LIN {X 0,Y 249.049,Z 231.079,A -85,B 0,C 180,E1 -18869.473,E2 -18869.473} C_VEL
LIN {X 0,Y 249.067,Z 231.077,A -85,B 0,C 180,E1 -18873.162,E2 -18873.162} C_VEL
LIN {X 0,Y 249.056,Z 231.062,A -85,B 0,C 180,E1 -18876.73,E2 -18876.73} C_VEL
LIN {X 0,Y 249.103,Z 231.062,A -85,B 0,C 180,E1 -18880.211,E2 -18880.211} C_VEL
LIN {X 0,Y 249.237,Z 231.055,A -85,B 0,C 180,E1 -18883.622,E2 -18883.622} C_VEL
LIN {X 0,Y 249.239,Z 231.06,A -85,B 0,C 180,E1 -18888.616,E2 -18888.616} C_VEL
LIN {X 0,Y 249.449,Z 231.028,A -85,B 0,C 180,E1 -18891.902,E2 -18891.902} C_VEL
LIN {X 0,Y 249.291,Z 231.049,A -85,B 0,C 180,E1 -18895.149,E2 -18895.149} C_VEL
LIN {X 0,Y 249.671,Z 231.01,A -85,B 0,C 180,E1 -18898.387,E2 -18898.387} C_VEL
LIN {X 0,Y 249.671,Z 231.008,A -85,B 0,C 180,E1 -18901.613,E2 -18901.613} C_VEL
LIN {X 0,Y 249.436,Z 231.036,A -85,B 0,C 180,E1 -18906.714,E2 -18906.714} C_VEL
LIN {X 0,Y 249.339,Z 231.046,A -85,B 0,C 180,E1 -18909.737,E2 -18909.737} C_VEL
LIN {X 0,Y 249.192,Z 231.07,A -85,B 0,C 180,E1 -18914.704,E2 -18914.704} C_VEL
LIN {X 0,Y 249.13,Z 231.075,A -85,B 0,C 180,E1 -18918.078,E2 -18918.078} C_VEL
LIN {X 0,Y 249.08,Z 231.078,A -85,B 0,C 180,E1 -18921.519,E2 -18921.519} C_VEL
LIN {X 0,Y 249.113,Z 231.045,A -85,B 0,C 180,E1 -18925.476,E2 -18925.476} C_VEL
LIN {X 0,Y 249.08,Z 231.083,A -85,B 0,C 180,E1 -18928.994,E2 -18928.994} C_VEL
LIN {X 0,Y 249.027,Z 231.091,A -85,B 0,C 180,E1 -18932.427,E2 -18932.427} C_VEL
LIN {X 0,Y 249.027,Z 231.083,A -85,B 0,C 180,E1 -18936.346,E2 -18936.346} C_VEL
LIN {X 0,Y 249.031,Z 231.1,A -85,B 0,C 180,E1 -18939.615,E2 -18939.615} C_VEL
LIN {X 0,Y 249.908,Z 233.771,A -85,B 0,C 180,E1 -18939.977,E2 -18939.977} C_VEL
LIN {X 0,Y 251.817,Z 235.917,A -85,B 0,C 180,E1 -18940.589,E2 -18940.589} C_VEL
LIN {X 0,Y 252.607,Z 236.622,A -85,B 0,C 180,E1 -18940.83,E2 -18940.83} C_VEL
LIN {X 0,Y 254.612,Z 239.846,A -85,B 0,C 180,E1 -18941.489,E2 -18941.489} C_VEL
LIN {X 0,Y 256.321,Z 241.907,A -85,B 0,C 180,E1 -18942.007,E2 -18942.007} C_VEL
LIN {X 0,Y 263.064,Z 251.483,A -85,B 0,C 180,E1 -18943.997,E2 -18943.997} C_VEL
LIN {X 0,Y 271.116,Z 263.635,A -85,B 0,C 180,E1 -18946.185,E2 -18946.185} C_VEL
LIN {X 0,Y 276.17,Z 272.352,A -85,B 0,C 180,E1 -18947.494,E2 -18947.494} C_VEL
LIN {X 0,Y 283.771,Z 287.993,A -85,B 0,C 180,E1 -18949.41,E2 -18949.41} C_VEL
LIN {X 0,Y 285.944,Z 292.88,A -85,B 0,C 180,E1 -18949.943,E2 -18949.943} C_VEL
LIN {X 0,Y 281.183,Z 391.143,A -85,B 0,C 180,E1 -18952.354,E2 -18952.354} C_VEL
LIN {X 0,Y 279.713,Z 406.301,A -85,B 0,C 180,E1 -18952.971,E2 -18952.971} C_VEL
LIN {X 0,Y 277.742,Z 421.037,A -85,B 0,C 180,E1 -18953.851,E2 -18953.851} C_VEL
LIN {X 0,Y 275.453,Z 434.469,A -85,B 0,C 180,E1 -18954.923,E2 -18954.923} C_VEL
LIN {X 0,Y 272.602,Z 448.403,A -85,B 0,C 180,E1 -18956.339,E2 -18956.339} C_VEL
LIN {X 0,Y 269.202,Z 462.16,A -85,B 0,C 180,E1 -18958.086,E2 -18958.086} C_VEL
LIN {X 0,Y 265.716,Z 474.57,A -85,B 0,C 180,E1 -18960.052,E2 -18960.052} C_VEL
LIN {X 0,Y 262.08,Z 486.635,A -85,B 0,C 180,E1 -18962.425,E2 -18962.425} C_VEL
LIN {X 0,Y 259.029,Z 496.066,A -85,B 0,C 180,E1 -18964.702,E2 -18964.702} C_VEL
LIN {X 0,Y 255.946,Z 505.251,A -85,B 0,C 180,E1 -18967.393,E2 -18967.393} C_VEL
LIN {X 0,Y 253.293,Z 512.885,A -85,B 0,C 180,E1 -18970.13,E2 -18970.13} C_VEL
LIN {X 0,Y 251.278,Z 519.21,A -85,B 0,C 180,E1 -18972.922,E2 -18972.922} C_VEL
LIN {X 0,Y 249.388,Z 525.021,A -85,B 0,C 180,E1 -18976.141,E2 -18976.141} C_VEL
LIN {X 0,Y 248.464,Z 528.456,A -85,B 0,C 180,E1 -18978.58,E2 -18978.58} C_VEL
LIN {X 0,Y 247.631,Z 531.932,A -85,B 0,C 180,E1 -18981.842,E2 -18981.842} C_VEL
LIN {X 0,Y 247.133,Z 534.228,A -85,B 0,C 180,E1 -18985.106,E2 -18985.106} C_VEL
LIN {X 0,Y 246.994,Z 535.396,A -85,B 0,C 180,E1 -18988.37,E2 -18988.37} C_VEL
LIN {X 0,Y 246.994,Z 535.409,A -85,B 0,C 180,E1 -18991.63,E2 -18991.63} C_VEL
LIN {X 0,Y 247.119,Z 534.293,A -85,B 0,C 180,E1 -18994.894,E2 -18994.894} C_VEL
LIN {X 0,Y 247.576,Z 532.048,A -85,B 0,C 180,E1 -18998.16,E2 -18998.16} C_VEL
LIN {X 0,Y 248.444,Z 528.617,A -85,B 0,C 180,E1 -19001.421,E2 -19001.421} C_VEL
LIN {X 0,Y 249.789,Z 523.917,A -85,B 0,C 180,E1 -19004.668,E2 -19004.668} C_VEL
LIN {X 0,Y 251.756,Z 517.821,A -85,B 0,C 180,E1 -19007.883,E2 -19007.883} C_VEL
LIN {X 0,Y 254.323,Z 510.141,A -85,B 0,C 180,E1 -19011.053,E2 -19011.053} C_VEL
LIN {X 0,Y 257.145,Z 501.947,A -85,B 0,C 180,E1 -19013.773,E2 -19013.773} C_VEL
LIN {X 0,Y 260.503,Z 492.069,A -85,B 0,C 180,E1 -19016.432,E2 -19016.432} C_VEL
LIN {X 0,Y 263.568,Z 481.946,A -85,B 0,C 180,E1 -19018.683,E2 -19018.683} C_VEL
LIN {X 0,Y 267.203,Z 469.879,A -85,B 0,C 180,E1 -19020.856,E2 -19020.856} C_VEL
LIN {X 0,Y 270.381,Z 457.778,A -85,B 0,C 180,E1 -19022.639,E2 -19022.639} C_VEL
LIN {X 0,Y 273.52,Z 444.619,A -85,B 0,C 180,E1 -19024.198,E2 -19024.198} C_VEL
LIN {X 0,Y 276.054,Z 431.618,A -85,B 0,C 180,E1 -19025.444,E2 -19025.444} C_VEL
LIN {X 0,Y 278.359,Z 417.38,A -85,B 0,C 180,E1 -19026.505,E2 -19026.505} C_VEL
LIN {X 0,Y 280.223,Z 402.085,A -85,B 0,C 180,E1 -19027.345,E2 -19027.345} C_VEL
LIN {X 0,Y 281.549,Z 387.286,A -85,B 0,C 180,E1 -19027.871,E2 -19027.871} C_VEL
LIN {X 0,Y 285.265,Z 308.817,A -85,B 0,C 180,E1 -19029.794,E2 -19029.794} C_VEL
LIN {X 0,Y 286.039,Z 293.023,A -85,B 0,C 180,E1 -19030.172,E2 -19030.172} C_VEL
LIN {X 0,Y 278.243,Z 276.265,A -85,B 0,C 180,E1 -19032.12,E2 -19032.12} C_VEL
LIN {X 0,Y 272.879,Z 266.444,A -85,B 0,C 180,E1 -19033.502,E2 -19033.502} C_VEL
LIN {X 0,Y 264.325,Z 253.238,A -85,B 0,C 180,E1 -19035.804,E2 -19035.804} C_VEL
LIN {X 0,Y 258.155,Z 244.549,A -85,B 0,C 180,E1 -19037.59,E2 -19037.59} C_VEL
LIN {X 0,Y 255.32,Z 240.562,A -85,B 0,C 180,E1 -19038.462,E2 -19038.462} C_VEL
LIN {X 0,Y 253.026,Z 237.492,A -85,B 0,C 180,E1 -19039.186,E2 -19039.186} C_VEL
LIN {X 0,Y 252.167,Z 236.141,A -85,B 0,C 180,E1 -19039.472,E2 -19039.472} C_VEL
LIN {X 0,Y 250.104,Z 234.024,A -85,B 0,C 180,E1 -19040.125,E2 -19040.125} C_VEL
LIN {X 0,Y 249.181,Z 231.839,A -85,B 0,C 180,E1 -19040.479,E2 -19040.479} C_VEL
LIN {X 0,Y 249.031,Z 231.081,A -85,B 0,C 180,E1 -19040.581,E2 -19040.581} C_VEL
LIN {X 0,Y 249.071,Z 231.082,A -85,B 0,C 180,E1 -19044.912,E2 -19044.912} C_VEL
LIN {X 0,Y 249.048,Z 231.057,A -85,B 0,C 180,E1 -19049.472,E2 -19049.472} C_VEL
LIN {X 0,Y 249.07,Z 231.077,A -85,B 0,C 180,E1 -19053.162,E2 -19053.162} C_VEL
LIN {X 0,Y 249.075,Z 231.077,A -85,B 0,C 180,E1 -19056.732,E2 -19056.732} C_VEL
LIN {X 0,Y 249.093,Z 231.077,A -85,B 0,C 180,E1 -19059.999,E2 -19059.999} C_VEL
LIN {X 0,Y 248.488,Z 231.159,A -85,B 0,C 180,E1 -19061.349,E2 -19061.349} C_VEL
LIN {X 0,Y 245.681,Z 231.508,A -85,B 0,C 180,E1 -19063.553,E2 -19063.553} C_VEL
LIN {X 0,Y 243.262,Z 231.8,A -85,B 0,C 180,E1 -19065.347,E2 -19065.347} C_VEL
LIN {X 0,Y 242.224,Z 231.929,A -85,B 0,C 180,E1 -19066.739,E2 -19066.739} C_VEL
LIN {X 0,Y 242.141,Z 231.939,A -85,B 0,C 180,E1 -19067.21,E2 -19067.21} C_VEL
LIN {X 0,Y 242.421,Z 231.909,A -85,B 0,C 180,E1 -19071.665,E2 -19071.665} C_VEL
LIN {X 0,Y 242.252,Z 231.921,A -85,B 0,C 180,E1 -19075.007,E2 -19075.007} C_VEL
LIN {X 0,Y 242.631,Z 231.879,A -85,B 0,C 180,E1 -19078.34,E2 -19078.34} C_VEL
LIN {X 0,Y 242.631,Z 231.887,A -85,B 0,C 180,E1 -19081.66,E2 -19081.66} C_VEL
LIN {X 0,Y 242.418,Z 231.914,A -85,B 0,C 180,E1 -19086.659,E2 -19086.659} C_VEL
LIN {X 0,Y 242.262,Z 231.931,A -85,B 0,C 180,E1 -19090.024,E2 -19090.024} C_VEL
LIN {X 0,Y 242.151,Z 231.951,A -85,B 0,C 180,E1 -19095.142,E2 -19095.142} C_VEL
LIN {X 0,Y 242.066,Z 231.954,A -85,B 0,C 180,E1 -19098.624,E2 -19098.624} C_VEL
LIN {X 0,Y 242.008,Z 231.957,A -85,B 0,C 180,E1 -19102.18,E2 -19102.18} C_VEL
LIN {X 0,Y 242.062,Z 231.949,A -85,B 0,C 180,E1 -19105.838,E2 -19105.838} C_VEL
LIN {X 0,Y 242.026,Z 231.964,A -85,B 0,C 180,E1 -19109.58,E2 -19109.58} C_VEL
LIN {X 0,Y 241.984,Z 231.959,A -85,B 0,C 180,E1 -19113.492,E2 -19113.492} C_VEL
LIN {X 0,Y 242.033,Z 232.067,A -85,B 0,C 180,E1 -19115.733,E2 -19115.733} C_VEL
LIN {X 0,Y 243.179,Z 235.576,A -85,B 0,C 180,E1 -19117.587,E2 -19117.587} C_VEL
LIN {X 0,Y 246.165,Z 240.122,A -85,B 0,C 180,E1 -19118.683,E2 -19118.683} C_VEL
LIN {X 0,Y 248.537,Z 243.621,A -85,B 0,C 180,E1 -19119.512,E2 -19119.512} C_VEL
LIN {X 0,Y 251.759,Z 248.527,A -85,B 0,C 180,E1 -19120.598,E2 -19120.598} C_VEL
LIN {X 0,Y 257.901,Z 258.318,A -85,B 0,C 180,E1 -19122.551,E2 -19122.551} C_VEL
LIN {X 0,Y 265.034,Z 270.727,A -85,B 0,C 180,E1 -19124.664,E2 -19124.664} C_VEL
LIN {X 0,Y 272.169,Z 284.843,A -85,B 0,C 180,E1 -19126.657,E2 -19126.657} C_VEL
LIN {X 0,Y 278.428,Z 298.931,A -85,B 0,C 180,E1 -19128.331,E2 -19128.331} C_VEL
LIN {X 0,Y 280.219,Z 303.302,A -85,B 0,C 180,E1 -19128.799,E2 -19128.799} C_VEL
LIN {X 0,Y 275.303,Z 401.477,A -85,B 0,C 180,E1 -19131.228,E2 -19131.228} C_VEL
LIN {X 0,Y 273.864,Z 416.504,A -85,B 0,C 180,E1 -19131.809,E2 -19131.809} C_VEL
LIN {X 0,Y 271.576,Z 431.908,A -85,B 0,C 180,E1 -19132.662,E2 -19132.662} C_VEL
LIN {X 0,Y 268.904,Z 446.169,A -85,B 0,C 180,E1 -19133.75,E2 -19133.75} C_VEL
LIN {X 0,Y 265.932,Z 459.788,A -85,B 0,C 180,E1 -19135.109,E2 -19135.109} C_VEL
LIN {X 0,Y 262.541,Z 472.752,A -85,B 0,C 180,E1 -19136.718,E2 -19136.718} C_VEL
LIN {X 0,Y 258.73,Z 485.615,A -85,B 0,C 180,E1 -19138.702,E2 -19138.702} C_VEL
LIN {X 0,Y 255.333,Z 496.392,A -85,B 0,C 180,E1 -19140.754,E2 -19140.754} C_VEL
LIN {X 0,Y 251.961,Z 506.52,A -85,B 0,C 180,E1 -19143.093,E2 -19143.093} C_VEL
LIN {X 0,Y 248.794,Z 516.14,A -85,B 0,C 180,E1 -19145.821,E2 -19145.821} C_VEL
LIN {X 0,Y 245.939,Z 524.293,A -85,B 0,C 180,E1 -19148.633,E2 -19148.633} C_VEL
LIN {X 0,Y 243.714,Z 531.043,A -85,B 0,C 180,E1 -19151.506,E2 -19151.506} C_VEL
LIN {X 0,Y 241.835,Z 537.282,A -85,B 0,C 180,E1 -19154.838,E2 -19154.838} C_VEL
LIN {X 0,Y 240.568,Z 542.112,A -85,B 0,C 180,E1 -19158.2,E2 -19158.2} C_VEL
LIN {X 0,Y 239.938,Z 545.658,A -85,B 0,C 180,E1 -19161.579,E2 -19161.579} C_VEL
LIN {X 0,Y 239.734,Z 548.194,A -85,B 0,C 180,E1 -19165.367,E2 -19165.367} C_VEL
LIN {X 0,Y 239.828,Z 549.172,A -85,B 0,C 180,E1 -19168.321,E2 -19168.321} C_VEL
LIN {X 0,Y 239.89,Z 549.328,A -85,B 0,C 180,E1 -19170,E2 -19170} C_VEL
LIN {X 0,Y 239.743,Z 548.713,A -85,B 0,C 180,E1 -19173.361,E2 -19173.361} C_VEL
LIN {X 0,Y 239.785,Z 546.943,A -85,B 0,C 180,E1 -19176.733,E2 -19176.733} C_VEL
LIN {X 0,Y 240.221,Z 543.999,A -85,B 0,C 180,E1 -19180.11,E2 -19180.11} C_VEL
LIN {X 0,Y 241.155,Z 539.813,A -85,B 0,C 180,E1 -19183.482,E2 -19183.482} C_VEL
LIN {X 0,Y 242.59,Z 534.273,A -85,B 0,C 180,E1 -19186.84,E2 -19186.84} C_VEL
LIN {X 0,Y 244.888,Z 527.241,A -85,B 0,C 180,E1 -19190.144,E2 -19190.144} C_VEL
LIN {X 0,Y 247.897,Z 518.5,A -85,B 0,C 180,E1 -19193.384,E2 -19193.384} C_VEL
LIN {X 0,Y 250.77,Z 509.884,A -85,B 0,C 180,E1 -19195.993,E2 -19195.993} C_VEL
LIN {X 0,Y 254.158,Z 499.789,A -85,B 0,C 180,E1 -19198.489,E2 -19198.489} C_VEL
LIN {X 0,Y 258.085,Z 487.563,A -85,B 0,C 180,E1 -19200.929,E2 -19200.929} C_VEL
LIN {X 0,Y 261.814,Z 475.101,A -85,B 0,C 180,E1 -19202.927,E2 -19202.927} C_VEL
LIN {X 0,Y 265.217,Z 462.341,A -85,B 0,C 180,E1 -19204.579,E2 -19204.579} C_VEL
LIN {X 0,Y 268.483,Z 447.763,A -85,B 0,C 180,E1 -19206.083,E2 -19206.083} C_VEL
LIN {X 0,Y 271.288,Z 432.708,A -85,B 0,C 180,E1 -19207.268,E2 -19207.268} C_VEL
LIN {X 0,Y 273.573,Z 417.629,A -85,B 0,C 180,E1 -19208.122,E2 -19208.122} C_VEL
LIN {X 0,Y 275.209,Z 401.795,A -85,B 0,C 180,E1 -19208.729,E2 -19208.729} C_VEL
LIN {X 0,Y 280.138,Z 304.198,A -85,B 0,C 180,E1 -19211.137,E2 -19211.137} C_VEL
LIN {X 0,Y 279.83,Z 302.568,A -85,B 0,C 180,E1 -19211.246,E2 -19211.246} C_VEL
LIN {X 0,Y 273.425,Z 287.591,A -85,B 0,C 180,E1 -19212.947,E2 -19212.947} C_VEL
LIN {X 0,Y 266.338,Z 273.301,A -85,B 0,C 180,E1 -19214.9,E2 -19214.9} C_VEL
LIN {X 0,Y 259.58,Z 261.145,A -85,B 0,C 180,E1 -19216.872,E2 -19216.872} C_VEL
LIN {X 0,Y 253.119,Z 250.672,A -85,B 0,C 180,E1 -19218.884,E2 -19218.884} C_VEL
LIN {X 0,Y 250.005,Z 245.759,A -85,B 0,C 180,E1 -19219.915,E2 -19219.915} C_VEL
LIN {X 0,Y 246.157,Z 240.034,A -85,B 0,C 180,E1 -19221.242,E2 -19221.242} C_VEL
LIN {X 0,Y 243.216,Z 235.593,A -85,B 0,C 180,E1 -19222.315,E2 -19222.315} C_VEL
LIN {X 0,Y 242.038,Z 231.948,A -85,B 0,C 180,E1 -19224.268,E2 -19224.268} C_VEL
LIN {X 0,Y 241.974,Z 231.964,A -85,B 0,C 180,E1 -19228.48,E2 -19228.48} C_VEL
LIN {X 0,Y 242.005,Z 231.96,A -85,B 0,C 180,E1 -19232.313,E2 -19232.313} C_VEL
LIN {X 0,Y 242.036,Z 231.948,A -85,B 0,C 180,E1 -19236.014,E2 -19236.014} C_VEL
LIN {X 0,Y 242.03,Z 231.933,A -85,B 0,C 180,E1 -19239.608,E2 -19239.608} C_VEL
LIN {X 0,Y 242.159,Z 231.938,A -85,B 0,C 180,E1 -19243.278,E2 -19243.278} C_VEL
LIN {X 0,Y 242.175,Z 231.936,A -85,B 0,C 180,E1 -19248.279,E2 -19248.279} C_VEL
LIN {X 0,Y 242.395,Z 231.906,A -85,B 0,C 180,E1 -19251.665,E2 -19251.665} C_VEL
LIN {X 0,Y 242.251,Z 231.926,A -85,B 0,C 180,E1 -19255.007,E2 -19255.007} C_VEL
LIN {X 0,Y 242.631,Z 231.887,A -85,B 0,C 180,E1 -19258.34,E2 -19258.34} C_VEL
LIN {X 0,Y 242.631,Z 231.885,A -85,B 0,C 180,E1 -19261.66,E2 -19261.66} C_VEL
LIN {X 0,Y 242.417,Z 231.914,A -85,B 0,C 180,E1 -19266.685,E2 -19266.685} C_VEL
LIN {X 0,Y 242.263,Z 231.93,A -85,B 0,C 180,E1 -19270.024,E2 -19270.024} C_VEL
LIN {X 0,Y 242.152,Z 231.947,A -85,B 0,C 180,E1 -19275.142,E2 -19275.142} C_VEL
LIN {X 0,Y 242.065,Z 231.958,A -85,B 0,C 180,E1 -19278.625,E2 -19278.625} C_VEL
LIN {X 0,Y 242.002,Z 231.965,A -85,B 0,C 180,E1 -19282.181,E2 -19282.181} C_VEL
LIN {X 0,Y 242.063,Z 231.921,A -85,B 0,C 180,E1 -19285.839,E2 -19285.839} C_VEL
LIN {X 0,Y 242.027,Z 231.963,A -85,B 0,C 180,E1 -19289.581,E2 -19289.581} C_VEL
LIN {X 0,Y 241.977,Z 231.962,A -85,B 0,C 180,E1 -19293.493,E2 -19293.493} C_VEL
LIN {X 0,Y 241.993,Z 231.968,A -85,B 0,C 180,E1 -19297.582,E2 -19297.582} C_VEL
LIN {X 0,Y 242.872,Z 234.562,A -85,B 0,C 180,E1 -19297.975,E2 -19297.975} C_VEL
LIN {X 0,Y 244.641,Z 236.655,A -85,B 0,C 180,E1 -19298.604,E2 -19298.604} C_VEL
LIN {X 0,Y 245.767,Z 237.766,A -85,B 0,C 180,E1 -19298.985,E2 -19298.985} C_VEL
LIN {X 0,Y 247.872,Z 241.021,A -85,B 0,C 180,E1 -19299.733,E2 -19299.733} C_VEL
LIN {X 0,Y 249.478,Z 242.818,A -85,B 0,C 180,E1 -19300.257,E2 -19300.257} C_VEL
LIN {X 0,Y 252.08,Z 246.354,A -85,B 0,C 180,E1 -19301.107,E2 -19301.107} C_VEL
LIN {X 0,Y 259.473,Z 256.984,A -85,B 0,C 180,E1 -19303.381,E2 -19303.381} C_VEL
LIN {X 0,Y 267.601,Z 269.403,A -85,B 0,C 180,E1 -19305.666,E2 -19305.666} C_VEL
LIN {X 0,Y 272.473,Z 278.147,A -85,B 0,C 180,E1 -19306.977,E2 -19306.977} C_VEL
LIN {X 0,Y 279.378,Z 292.763,A -85,B 0,C 180,E1 -19308.788,E2 -19308.788} C_VEL
LIN {X 0,Y 280.418,Z 295.109,A -85,B 0,C 180,E1 -19309.053,E2 -19309.053} C_VEL
LIN {X 0,Y 278.39,Z 336.907,A -85,B 0,C 180,E1 -19310.083,E2 -19310.083} C_VEL
LIN {X 0,Y 275.611,Z 391.359,A -85,B 0,C 180,E1 -19311.455,E2 -19311.455} C_VEL
LIN {X 0,Y 274.097,Z 406.512,A -85,B 0,C 180,E1 -19312.08,E2 -19312.08} C_VEL
LIN {X 0,Y 272.04,Z 421.246,A -85,B 0,C 180,E1 -19312.969,E2 -19312.969} C_VEL
LIN {X 0,Y 269.699,Z 434.359,A -85,B 0,C 180,E1 -19314.023,E2 -19314.023} C_VEL
LIN {X 0,Y 266.729,Z 448.609,A -85,B 0,C 180,E1 -19315.494,E2 -19315.494} C_VEL
LIN {X 0,Y 263.202,Z 462.366,A -85,B 0,C 180,E1 -19317.269,E2 -19317.269} C_VEL
LIN {X 0,Y 259.597,Z 474.775,A -85,B 0,C 180,E1 -19319.27,E2 -19319.27} C_VEL
LIN {X 0,Y 256.058,Z 485.733,A -85,B 0,C 180,E1 -19321.438,E2 -19321.438} C_VEL
LIN {X 0,Y 253.169,Z 494.792,A -85,B 0,C 180,E1 -19323.631,E2 -19323.631} C_VEL
LIN {X 0,Y 249.824,Z 504.233,A -85,B 0,C 180,E1 -19326.368,E2 -19326.368} C_VEL
LIN {X 0,Y 246.978,Z 512.088,A -85,B 0,C 180,E1 -19329.164,E2 -19329.164} C_VEL
LIN {X 0,Y 244.447,Z 519.414,A -85,B 0,C 180,E1 -19332.43,E2 -19332.43} C_VEL
LIN {X 0,Y 242.476,Z 525.224,A -85,B 0,C 180,E1 -19335.738,E2 -19335.738} C_VEL
LIN {X 0,Y 241.493,Z 528.658,A -85,B 0,C 180,E1 -19338.246,E2 -19338.246} C_VEL
LIN {X 0,Y 240.602,Z 532.133,A -85,B 0,C 180,E1 -19341.602,E2 -19341.602} C_VEL
LIN {X 0,Y 240.058,Z 534.429,A -85,B 0,C 180,E1 -19344.961,E2 -19344.961} C_VEL
LIN {X 0,Y 239.907,Z 535.597,A -85,B 0,C 180,E1 -19348.321,E2 -19348.321} C_VEL
LIN {X 0,Y 239.906,Z 535.609,A -85,B 0,C 180,E1 -19351.679,E2 -19351.679} C_VEL
LIN {X 0,Y 240.058,Z 534.494,A -85,B 0,C 180,E1 -19355.039,E2 -19355.039} C_VEL
LIN {X 0,Y 240.523,Z 532.249,A -85,B 0,C 180,E1 -19358.401,E2 -19358.401} C_VEL
LIN {X 0,Y 241.459,Z 528.818,A -85,B 0,C 180,E1 -19361.756,E2 -19361.756} C_VEL
LIN {X 0,Y 242.912,Z 524.117,A -85,B 0,C 180,E1 -19365.093,E2 -19365.093} C_VEL
LIN {X 0,Y 244.989,Z 518.021,A -85,B 0,C 180,E1 -19368.394,E2 -19368.394} C_VEL
LIN {X 0,Y 247.664,Z 510.341,A -85,B 0,C 180,E1 -19371.647,E2 -19371.647} C_VEL
LIN {X 0,Y 250.641,Z 502.146,A -85,B 0,C 180,E1 -19374.43,E2 -19374.43} C_VEL
LIN {X 0,Y 254.126,Z 492.269,A -85,B 0,C 180,E1 -19377.149,E2 -19377.149} C_VEL
LIN {X 0,Y 257.344,Z 482.145,A -85,B 0,C 180,E1 -19379.443,E2 -19379.443} C_VEL
LIN {X 0,Y 261.124,Z 470.076,A -85,B 0,C 180,E1 -19381.656,E2 -19381.656} C_VEL
LIN {X 0,Y 264.427,Z 457.974,A -85,B 0,C 180,E1 -19383.469,E2 -19383.469} C_VEL
LIN {X 0,Y 267.679,Z 444.815,A -85,B 0,C 180,E1 -19385.052,E2 -19385.052} C_VEL
LIN {X 0,Y 270.322,Z 431.776,A -85,B 0,C 180,E1 -19386.318,E2 -19386.318} C_VEL
LIN {X 0,Y 272.686,Z 417.572,A -85,B 0,C 180,E1 -19387.392,E2 -19387.392} C_VEL
LIN {X 0,Y 274.636,Z 402.272,A -85,B 0,C 180,E1 -19388.239,E2 -19388.239} C_VEL
LIN {X 0,Y 276.001,Z 387.466,A -85,B 0,C 180,E1 -19388.773,E2 -19388.773} C_VEL
LIN {X 0,Y 279.829,Z 309.551,A -85,B 0,C 180,E1 -19390.709,E2 -19390.709} C_VEL
LIN {X 0,Y 280.529,Z 295.264,A -85,B 0,C 180,E1 -19391.06,E2 -19391.06} C_VEL
LIN {X 0,Y 273.252,Z 279.606,A -85,B 0,C 180,E1 -19392.961,E2 -19392.961} C_VEL
LIN {X 0,Y 268.612,Z 271.045,A -85,B 0,C 180,E1 -19394.209,E2 -19394.209} C_VEL
LIN {X 0,Y 260.421,Z 258.255,A -85,B 0,C 180,E1 -19396.502,E2 -19396.502} C_VEL
LIN {X 0,Y 254.1,Z 249.275,A -85,B 0,C 180,E1 -19398.409,E2 -19398.409} C_VEL
LIN {X 0,Y 251.874,Z 246.083,A -85,B 0,C 180,E1 -19399.123,E2 -19399.123} C_VEL
LIN {X 0,Y 249.252,Z 242.356,A -85,B 0,C 180,E1 -19399.993,E2 -19399.993} C_VEL
LIN {X 0,Y 246.59,Z 239.269,A -85,B 0,C 180,E1 -19400.88,E2 -19400.88} C_VEL
LIN {X 0,Y 245.42,Z 237.185,A -85,B 0,C 180,E1 -19401.315,E2 -19401.315} C_VEL
LIN {X 0,Y 243.267,Z 235.184,A -85,B 0,C 180,E1 -19402.052,E2 -19402.052} C_VEL
LIN {X 0,Y 242.149,Z 232.717,A -85,B 0,C 180,E1 -19402.512,E2 -19402.512} C_VEL
LIN {X 0,Y 241.999,Z 231.937,A -85,B 0,C 180,E1 -19402.682,E2 -19402.682} C_VEL
LIN {X 0,Y 241.988,Z 231.951,A -85,B 0,C 180,E1 -19406.508,E2 -19406.508} C_VEL
LIN {X 0,Y 242.034,Z 231.945,A -85,B 0,C 180,E1 -19410.586,E2 -19410.586} C_VEL
LIN {X 0,Y 242.064,Z 231.949,A -85,B 0,C 180,E1 -19414.182,E2 -19414.182} C_VEL
LIN {X 0,Y 242.049,Z 231.952,A -85,B 0,C 180,E1 -19418.297,E2 -19418.297} C_VEL
LIN {X 0,Y 242.159,Z 231.946,A -85,B 0,C 180,E1 -19423.278,E2 -19423.278} C_VEL
LIN {X 0,Y 242.141,Z 231.939,A -85,B 0,C 180,E1 -19427.21,E2 -19427.21} C_VEL
LIN {X 0,Y 241.504,Z 232.026,A -85,B 0,C 180,E1 -19428.601,E2 -19428.601} C_VEL
LIN {X 0,Y 238.751,Z 232.366,A -85,B 0,C 180,E1 -19430.873,E2 -19430.873} C_VEL
LIN {X 0,Y 235.573,Z 232.759,A -85,B 0,C 180,E1 -19433.673,E2 -19433.673} C_VEL
LIN {X 0,Y 235.226,Z 232.796,A -85,B 0,C 180,E1 -19434.64,E2 -19434.64} C_VEL
LIN {X 0,Y 235.591,Z 232.756,A -85,B 0,C 180,E1 -19438.29,E2 -19438.29} C_VEL
LIN {X 0,Y 235.591,Z 232.764,A -85,B 0,C 180,E1 -19441.709,E2 -19441.709} C_VEL
LIN {X 0,Y 235.368,Z 232.791,A -85,B 0,C 180,E1 -19446.86,E2 -19446.86} C_VEL
LIN {X 0,Y 235.209,Z 232.812,A -85,B 0,C 180,E1 -19450.328,E2 -19450.328} C_VEL
LIN {X 0,Y 235.102,Z 232.829,A -85,B 0,C 180,E1 -19455.607,E2 -19455.607} C_VEL
LIN {X 0,Y 235.003,Z 232.842,A -85,B 0,C 180,E1 -19459.206,E2 -19459.206} C_VEL
LIN {X 0,Y 234.957,Z 232.841,A -85,B 0,C 180,E1 -19462.883,E2 -19462.883} C_VEL
LIN {X 0,Y 234.966,Z 232.837,A -85,B 0,C 180,E1 -19466.658,E2 -19466.658} C_VEL
LIN {X 0,Y 234.928,Z 232.846,A -85,B 0,C 180,E1 -19470.568,E2 -19470.568} C_VEL
LIN {X 0,Y 234.958,Z 233.014,A -85,B 0,C 180,E1 -19473.897,E2 -19473.897} C_VEL
LIN {X 0,Y 235.791,Z 235.407,A -85,B 0,C 180,E1 -19475.196,E2 -19475.196} C_VEL
LIN {X 0,Y 239.209,Z 240.287,A -85,B 0,C 180,E1 -19476.574,E2 -19476.574} C_VEL
LIN {X 0,Y 244.83,Z 248.51,A -85,B 0,C 180,E1 -19478.679,E2 -19478.679} C_VEL
LIN {X 0,Y 250.854,Z 257.928,A -85,B 0,C 180,E1 -19480.762,E2 -19480.762} C_VEL
LIN {X 0,Y 258.936,Z 271.679,A -85,B 0,C 180,E1 -19483.328,E2 -19483.328} C_VEL
LIN {X 0,Y 266.691,Z 286.936,A -85,B 0,C 180,E1 -19485.62,E2 -19485.62} C_VEL
LIN {X 0,Y 273.101,Z 301.379,A -85,B 0,C 180,E1 -19487.42,E2 -19487.42} C_VEL
LIN {X 0,Y 274.782,Z 305.409,A -85,B 0,C 180,E1 -19487.878,E2 -19487.878} C_VEL
LIN {X 0,Y 270.317,Z 393.45,A -85,B 0,C 180,E1 -19490.071,E2 -19490.071} C_VEL
LIN {X 0,Y 269.205,Z 408.552,A -85,B 0,C 180,E1 -19490.542,E2 -19490.542} C_VEL
LIN {X 0,Y 267.336,Z 423.536,A -85,B 0,C 180,E1 -19491.245,E2 -19491.245} C_VEL
LIN {X 0,Y 264.859,Z 437.611,A -85,B 0,C 180,E1 -19492.149,E2 -19492.149} C_VEL
LIN {X 0,Y 262.003,Z 451.527,A -85,B 0,C 180,E1 -19493.357,E2 -19493.357} C_VEL
LIN {X 0,Y 258.557,Z 465.591,A -85,B 0,C 180,E1 -19494.924,E2 -19494.924} C_VEL
LIN {X 0,Y 254.737,Z 478.702,A -85,B 0,C 180,E1 -19496.748,E2 -19496.748} C_VEL
LIN {X 0,Y 251.025,Z 490.536,A -85,B 0,C 180,E1 -19498.806,E2 -19498.806} C_VEL
LIN {X 0,Y 247.322,Z 501.384,A -85,B 0,C 180,E1 -19501.114,E2 -19501.114} C_VEL
LIN {X 0,Y 243.918,Z 511.073,A -85,B 0,C 180,E1 -19503.637,E2 -19503.637} C_VEL
LIN {X 0,Y 240.877,Z 519.634,A -85,B 0,C 180,E1 -19506.349,E2 -19506.349} C_VEL
LIN {X 0,Y 238.164,Z 527.139,A -85,B 0,C 180,E1 -19509.262,E2 -19509.262} C_VEL
LIN {X 0,Y 235.822,Z 534.146,A -85,B 0,C 180,E1 -19512.662,E2 -19512.662} C_VEL
LIN {X 0,Y 234.201,Z 539.663,A -85,B 0,C 180,E1 -19516.11,E2 -19516.11} C_VEL
LIN {X 0,Y 233.166,Z 543.839,A -85,B 0,C 180,E1 -19519.581,E2 -19519.581} C_VEL
LIN {X 0,Y 232.705,Z 546.772,A -85,B 0,C 180,E1 -19523.062,E2 -19523.062} C_VEL
LIN {X 0,Y 232.651,Z 548.525,A -85,B 0,C 180,E1 -19526.536,E2 -19526.536} C_VEL
LIN {X 0,Y 232.801,Z 549.127,A -85,B 0,C 180,E1 -19530,E2 -19530} C_VEL
LIN {X 0,Y 232.651,Z 548.511,A -85,B 0,C 180,E1 -19533.464,E2 -19533.464} C_VEL
LIN {X 0,Y 232.705,Z 546.741,A -85,B 0,C 180,E1 -19536.938,E2 -19536.938} C_VEL
LIN {X 0,Y 233.166,Z 543.795,A -85,B 0,C 180,E1 -19540.419,E2 -19540.419} C_VEL
LIN {X 0,Y 234.189,Z 539.609,A -85,B 0,C 180,E1 -19543.891,E2 -19543.891} C_VEL
LIN {X 0,Y 235.803,Z 533.785,A -85,B 0,C 180,E1 -19547.495,E2 -19547.495} C_VEL
LIN {X 0,Y 238.16,Z 527.037,A -85,B 0,C 180,E1 -19550.739,E2 -19550.739} C_VEL
LIN {X 0,Y 241.36,Z 518.297,A -85,B 0,C 180,E1 -19554.057,E2 -19554.057} C_VEL
LIN {X 0,Y 244.49,Z 509.269,A -85,B 0,C 180,E1 -19556.84,E2 -19556.84} C_VEL
LIN {X 0,Y 247.888,Z 499.584,A -85,B 0,C 180,E1 -19559.278,E2 -19559.278} C_VEL
LIN {X 0,Y 251.995,Z 487.358,A -85,B 0,C 180,E1 -19561.763,E2 -19561.763} C_VEL
LIN {X 0,Y 255.865,Z 474.896,A -85,B 0,C 180,E1 -19563.794,E2 -19563.794} C_VEL
LIN {X 0,Y 259.439,Z 461.812,A -85,B 0,C 180,E1 -19565.513,E2 -19565.513} C_VEL
LIN {X 0,Y 262.782,Z 447.556,A -85,B 0,C 180,E1 -19566.995,E2 -19566.995} C_VEL
LIN {X 0,Y 265.445,Z 433.76,A -85,B 0,C 180,E1 -19568.113,E2 -19568.113} C_VEL
LIN {X 0,Y 267.911,Z 418.318,A -85,B 0,C 180,E1 -19569.018,E2 -19569.018} C_VEL
LIN {X 0,Y 269.622,Z 403.033,A -85,B 0,C 180,E1 -19569.627,E2 -19569.627} C_VEL
LIN {X 0,Y 274.719,Z 305.584,A -85,B 0,C 180,E1 -19572.077,E2 -19572.077} C_VEL
LIN {X 0,Y 268.217,Z 290.233,A -85,B 0,C 180,E1 -19573.887,E2 -19573.887} C_VEL
LIN {X 0,Y 260.602,Z 274.912,A -85,B 0,C 180,E1 -19576.098,E2 -19576.098} C_VEL
LIN {X 0,Y 254.717,Z 264.543,A -85,B 0,C 180,E1 -19577.904,E2 -19577.904} C_VEL
LIN {X 0,Y 249.111,Z 255.283,A -85,B 0,C 180,E1 -19579.742,E2 -19579.742} C_VEL
LIN {X 0,Y 246.166,Z 250.607,A -85,B 0,C 180,E1 -19580.761,E2 -19580.761} C_VEL
LIN {X 0,Y 242.825,Z 245.511,A -85,B 0,C 180,E1 -19581.967,E2 -19581.967} C_VEL
LIN {X 0,Y 239.051,Z 240.03,A -85,B 0,C 180,E1 -19583.398,E2 -19583.398} C_VEL
LIN {X 0,Y 236.513,Z 236.451,A -85,B 0,C 180,E1 -19584.408,E2 -19584.408} C_VEL
LIN {X 0,Y 235.649,Z 235.075,A -85,B 0,C 180,E1 -19584.785,E2 -19584.785} C_VEL
LIN {X 0,Y 234.933,Z 232.837,A -85,B 0,C 180,E1 -19586.203,E2 -19586.203} C_VEL
LIN {X 0,Y 234.966,Z 232.831,A -85,B 0,C 180,E1 -19590.157,E2 -19590.157} C_VEL
LIN {X 0,Y 234.99,Z 232.831,A -85,B 0,C 180,E1 -19593.793,E2 -19593.793} C_VEL
LIN {X 0,Y 234.993,Z 232.803,A -85,B 0,C 180,E1 -19598.968,E2 -19598.968} C_VEL
LIN {X 0,Y 235.092,Z 232.819,A -85,B 0,C 180,E1 -19603.06,E2 -19603.06} C_VEL
LIN {X 0,Y 235.109,Z 232.815,A -85,B 0,C 180,E1 -19607.922,E2 -19607.922} C_VEL
LIN {X 0,Y 235.326,Z 232.787,A -85,B 0,C 180,E1 -19611.412,E2 -19611.412} C_VEL
LIN {X 0,Y 235.368,Z 232.79,A -85,B 0,C 180,E1 -19613.14,E2 -19613.14} C_VEL
LIN {X 0,Y 235.591,Z 232.764,A -85,B 0,C 180,E1 -19618.291,E2 -19618.291} C_VEL
LIN {X 0,Y 235.591,Z 232.762,A -85,B 0,C 180,E1 -19621.71,E2 -19621.71} C_VEL
LIN {X 0,Y 235.388,Z 232.79,A -85,B 0,C 180,E1 -19626.859,E2 -19626.859} C_VEL
LIN {X 0,Y 235.21,Z 232.811,A -85,B 0,C 180,E1 -19630.328,E2 -19630.328} C_VEL
LIN {X 0,Y 235.103,Z 232.822,A -85,B 0,C 180,E1 -19635.607,E2 -19635.607} C_VEL
LIN {X 0,Y 235.001,Z 232.837,A -85,B 0,C 180,E1 -19639.206,E2 -19639.206} C_VEL
LIN {X 0,Y 234.948,Z 232.844,A -85,B 0,C 180,E1 -19642.884,E2 -19642.884} C_VEL
LIN {X 0,Y 234.965,Z 232.806,A -85,B 0,C 180,E1 -19646.658,E2 -19646.658} C_VEL
LIN {X 0,Y 234.928,Z 232.84,A -85,B 0,C 180,E1 -19650.568,E2 -19650.568} C_VEL
LIN {X 0,Y 234.924,Z 232.84,A -85,B 0,C 180,E1 -19654.639,E2 -19654.639} C_VEL
LIN {X 0,Y 234.933,Z 232.896,A -85,B 0,C 180,E1 -19655.313,E2 -19655.313} C_VEL
LIN {X 0,Y 235.753,Z 235.339,A -85,B 0,C 180,E1 -19655.721,E2 -19655.721} C_VEL
LIN {X 0,Y 237.75,Z 237.648,A -85,B 0,C 180,E1 -19656.506,E2 -19656.506} C_VEL
LIN {X 0,Y 238.839,Z 238.529,A -85,B 0,C 180,E1 -19656.904,E2 -19656.904} C_VEL
LIN {X 0,Y 240.778,Z 241.715,A -85,B 0,C 180,E1 -19657.672,E2 -19657.672} C_VEL
LIN {X 0,Y 242.707,Z 243.819,A -85,B 0,C 180,E1 -19658.362,E2 -19658.362} C_VEL
LIN {X 0,Y 245.452,Z 247.542,A -85,B 0,C 180,E1 -19659.34,E2 -19659.34} C_VEL
LIN {X 0,Y 252.5,Z 257.33,A -85,B 0,C 180,E1 -19661.681,E2 -19661.681} C_VEL
LIN {X 0,Y 260.559,Z 269.535,A -85,B 0,C 180,E1 -19664.126,E2 -19664.126} C_VEL
LIN {X 0,Y 266.593,Z 279.634,A -85,B 0,C 180,E1 -19665.832,E2 -19665.832} C_VEL
LIN {X 0,Y 273.698,Z 294.412,A -85,B 0,C 180,E1 -19667.787,E2 -19667.787} C_VEL
LIN {X 0,Y 275.046,Z 297.6,A -85,B 0,C 180,E1 -19668.153,E2 -19668.153} C_VEL
LIN {X 0,Y 270.101,Z 391.575,A -85,B 0,C 180,E1 -19670.517,E2 -19670.517} C_VEL
LIN {X 0,Y 268.533,Z 406.724,A -85,B 0,C 180,E1 -19671.149,E2 -19671.149} C_VEL
LIN {X 0,Y 266.405,Z 421.455,A -85,B 0,C 180,E1 -19672.049,E2 -19672.049} C_VEL
LIN {X 0,Y 263.863,Z 435.241,A -85,B 0,C 180,E1 -19673.179,E2 -19673.179} C_VEL
LIN {X 0,Y 260.907,Z 448.816,A -85,B 0,C 180,E1 -19674.611,E2 -19674.611} C_VEL
LIN {X 0,Y 257.257,Z 462.571,A -85,B 0,C 180,E1 -19676.413,E2 -19676.413} C_VEL
LIN {X 0,Y 253.528,Z 474.979,A -85,B 0,C 180,E1 -19678.452,E2 -19678.452} C_VEL
LIN {X 0,Y 249.694,Z 486.38,A -85,B 0,C 180,E1 -19680.756,E2 -19680.756} C_VEL
LIN {X 0,Y 246.825,Z 494.995,A -85,B 0,C 180,E1 -19682.899,E2 -19682.899} C_VEL
LIN {X 0,Y 243.288,Z 504.437,A -85,B 0,C 180,E1 -19685.692,E2 -19685.692} C_VEL
LIN {X 0,Y 240.329,Z 512.291,A -85,B 0,C 180,E1 -19688.56,E2 -19688.56} C_VEL
LIN {X 0,Y 237.628,Z 519.618,A -85,B 0,C 180,E1 -19691.908,E2 -19691.908} C_VEL
LIN {X 0,Y 235.585,Z 525.426,A -85,B 0,C 180,E1 -19695.311,E2 -19695.311} C_VEL
LIN {X 0,Y 234.515,Z 528.861,A -85,B 0,C 180,E1 -19697.891,E2 -19697.891} C_VEL
LIN {X 0,Y 233.547,Z 532.336,A -85,B 0,C 180,E1 -19701.346,E2 -19701.346} C_VEL
LIN {X 0,Y 232.989,Z 534.631,A -85,B 0,C 180,E1 -19704.808,E2 -19704.808} C_VEL
LIN {X 0,Y 232.821,Z 535.797,A -85,B 0,C 180,E1 -19708.27,E2 -19708.27} C_VEL
LIN {X 0,Y 232.821,Z 535.81,A -85,B 0,C 180,E1 -19711.73,E2 -19711.73} C_VEL
LIN {X 0,Y 232.989,Z 534.565,A -85,B 0,C 180,E1 -19715.479,E2 -19715.479} C_VEL
LIN {X 0,Y 233.481,Z 532.45,A -85,B 0,C 180,E1 -19718.656,E2 -19718.656} C_VEL
LIN {X 0,Y 234.469,Z 529.019,A -85,B 0,C 180,E1 -19722.111,E2 -19722.111} C_VEL
LIN {X 0,Y 236.053,Z 524.317,A -85,B 0,C 180,E1 -19725.542,E2 -19725.542} C_VEL
LIN {X 0,Y 238.232,Z 518.221,A -85,B 0,C 180,E1 -19728.935,E2 -19728.935} C_VEL
LIN {X 0,Y 241.061,Z 510.54,A -85,B 0,C 180,E1 -19732.272,E2 -19732.272} C_VEL
LIN {X 0,Y 244.157,Z 502.346,A -85,B 0,C 180,E1 -19735.123,E2 -19735.123} C_VEL
LIN {X 0,Y 247.783,Z 492.468,A -85,B 0,C 180,E1 -19737.904,E2 -19737.904} C_VEL
LIN {X 0,Y 251.161,Z 482.343,A -85,B 0,C 180,E1 -19740.243,E2 -19740.243} C_VEL
LIN {X 0,Y 255.095,Z 470.274,A -85,B 0,C 180,E1 -19742.495,E2 -19742.495} C_VEL
LIN {X 0,Y 258.534,Z 458.171,A -85,B 0,C 180,E1 -19744.337,E2 -19744.337} C_VEL
LIN {X 0,Y 261.9,Z 445.01,A -85,B 0,C 180,E1 -19745.944,E2 -19745.944} C_VEL
LIN {X 0,Y 264.592,Z 432.235,A -85,B 0,C 180,E1 -19747.203,E2 -19747.203} C_VEL
LIN {X 0,Y 267.082,Z 417.764,A -85,B 0,C 180,E1 -19748.317,E2 -19748.317} C_VEL
LIN {X 0,Y 269.104,Z 402.461,A -85,B 0,C 180,E1 -19749.174,E2 -19749.174} C_VEL
LIN {X 0,Y 270.514,Z 387.647,A -85,B 0,C 180,E1 -19749.712,E2 -19749.712} C_VEL
LIN {X 0,Y 275.158,Z 298.383,A -85,B 0,C 180,E1 -19751.94,E2 -19751.94} C_VEL
LIN {X 0,Y 274.819,Z 296.927,A -85,B 0,C 180,E1 -19752.054,E2 -19752.054} C_VEL
LIN {X 0,Y 267.856,Z 281.938,A -85,B 0,C 180,E1 -19753.967,E2 -19753.967} C_VEL
LIN {X 0,Y 262.945,Z 273.244,A -85,B 0,C 180,E1 -19755.346,E2 -19755.346} C_VEL
LIN {X 0,Y 254.297,Z 259.894,A -85,B 0,C 180,E1 -19757.917,E2 -19757.917} C_VEL
LIN {X 0,Y 248.29,Z 251.4,A -85,B 0,C 180,E1 -19759.859,E2 -19759.859} C_VEL
LIN {X 0,Y 245.218,Z 247.285,A -85,B 0,C 180,E1 -19760.911,E2 -19760.911} C_VEL
LIN {X 0,Y 242.628,Z 243.605,A -85,B 0,C 180,E1 -19761.848,E2 -19761.848} C_VEL
LIN {X 0,Y 239.587,Z 239.963,A -85,B 0,C 180,E1 -19762.968,E2 -19762.968} C_VEL
LIN {X 0,Y 238.586,Z 238.134,A -85,B 0,C 180,E1 -19763.38,E2 -19763.38} C_VEL
LIN {X 0,Y 236.309,Z 236.162,A -85,B 0,C 180,E1 -19764.235,E2 -19764.235} C_VEL
LIN {X 0,Y 235.143,Z 233.752,A -85,B 0,C 180,E1 -19764.76,E2 -19764.76} C_VEL
LIN {X 0,Y 234.972,Z 232.836,A -85,B 0,C 180,E1 -19764.901,E2 -19764.901} C_VEL
LIN {X 0,Y 234.929,Z 232.813,A -85,B 0,C 180,E1 -19769.432,E2 -19769.432} C_VEL
LIN {X 0,Y 234.991,Z 232.829,A -85,B 0,C 180,E1 -19773.793,E2 -19773.793} C_VEL
LIN {X 0,Y 235.007,Z 232.835,A -85,B 0,C 180,E1 -19778.969,E2 -19778.969} C_VEL
LIN {X 0,Y 235.092,Z 232.824,A -85,B 0,C 180,E1 -19783.059,E2 -19783.059} C_VEL
LIN {X 0,Y 235.141,Z 232.82,A -85,B 0,C 180,E1 -19787.923,E2 -19787.923} C_VEL
LIN {X 0,Y 235.371,Z 232.784,A -85,B 0,C 180,E1 -19791.414,E2 -19791.414} C_VEL
LIN {X 0,Y 235.226,Z 232.796,A -85,B 0,C 180,E1 -19794.64,E2 -19794.64} C_VEL
LIN {X 0,Y 234.578,Z 232.885,A -85,B 0,C 180,E1 -19796.073,E2 -19796.073} C_VEL
LIN {X 0,Y 231.976,Z 233.216,A -85,B 0,C 180,E1 -19798.42,E2 -19798.42} C_VEL
LIN {X 0,Y 228.872,Z 233.602,A -85,B 0,C 180,E1 -19801.307,E2 -19801.307} C_VEL
LIN {X 0,Y 228.434,Z 233.649,A -85,B 0,C 180,E1 -19802.302,E2 -19802.302} C_VEL
LIN {X 0,Y 228.319,Z 233.667,A -85,B 0,C 180,E1 -19807.072,E2 -19807.072} C_VEL
LIN {X 0,Y 228.141,Z 233.695,A -85,B 0,C 180,E1 -19810.651,E2 -19810.651} C_VEL
LIN {X 0,Y 228.055,Z 233.699,A -85,B 0,C 180,E1 -19814.273,E2 -19814.273} C_VEL
LIN {X 0,Y 227.998,Z 233.701,A -85,B 0,C 180,E1 -19817.953,E2 -19817.953} C_VEL
LIN {X 0,Y 227.926,Z 233.712,A -85,B 0,C 180,E1 -19822.329,E2 -19822.329} C_VEL
LIN {X 0,Y 227.939,Z 233.712,A -85,B 0,C 180,E1 -19826.603,E2 -19826.603} C_VEL
LIN {X 0,Y 227.905,Z 233.721,A -85,B 0,C 180,E1 -19830.296,E2 -19830.296} C_VEL
LIN {X 0,Y 227.896,Z 233.758,A -85,B 0,C 180,E1 -19831.748,E2 -19831.748} C_VEL
LIN {X 0,Y 228.138,Z 234.874,A -85,B 0,C 180,E1 -19832.361,E2 -19832.361} C_VEL
LIN {X 0,Y 229.557,Z 237.459,A -85,B 0,C 180,E1 -19833.057,E2 -19833.057} C_VEL
LIN {X 0,Y 233.163,Z 241.68,A -85,B 0,C 180,E1 -19834.61,E2 -19834.61} C_VEL
LIN {X 0,Y 236.423,Z 246.308,A -85,B 0,C 180,E1 -19835.965,E2 -19835.965} C_VEL
LIN {X 0,Y 241.593,Z 254.107,A -85,B 0,C 180,E1 -19837.981,E2 -19837.981} C_VEL
LIN {X 0,Y 248.357,Z 265.084,A -85,B 0,C 180,E1 -19840.406,E2 -19840.406} C_VEL
LIN {X 0,Y 255.08,Z 276.751,A -85,B 0,C 180,E1 -19842.614,E2 -19842.614} C_VEL
LIN {X 0,Y 262.522,Z 291.692,A -85,B 0,C 180,E1 -19844.909,E2 -19844.909} C_VEL
LIN {X 0,Y 268.441,Z 305.273,A -85,B 0,C 180,E1 -19846.645,E2 -19846.645} C_VEL
LIN {X 0,Y 269.463,Z 307.846,A -85,B 0,C 180,E1 -19846.94,E2 -19846.94} C_VEL
LIN {X 0,Y 264.399,Z 401.113,A -85,B 0,C 180,E1 -19849.304,E2 -19849.304} C_VEL
LIN {X 0,Y 262.834,Z 416.124,A -85,B 0,C 180,E1 -19849.892,E2 -19849.892} C_VEL
LIN {X 0,Y 260.675,Z 430.221,A -85,B 0,C 180,E1 -19850.686,E2 -19850.686} C_VEL
LIN {X 0,Y 257.968,Z 443.786,A -85,B 0,C 180,E1 -19851.7,E2 -19851.7} C_VEL
LIN {X 0,Y 254.642,Z 458.179,A -85,B 0,C 180,E1 -19853.129,E2 -19853.129} C_VEL
LIN {X 0,Y 251.117,Z 471.061,A -85,B 0,C 180,E1 -19854.745,E2 -19854.745} C_VEL
LIN {X 0,Y 246.967,Z 484.144,A -85,B 0,C 180,E1 -19856.785,E2 -19856.785} C_VEL
LIN {X 0,Y 242.982,Z 495.994,A -85,B 0,C 180,E1 -19859.11,E2 -19859.11} C_VEL
LIN {X 0,Y 239.351,Z 505.969,A -85,B 0,C 180,E1 -19861.502,E2 -19861.502} C_VEL
LIN {X 0,Y 236.275,Z 514.48,A -85,B 0,C 180,E1 -19863.977,E2 -19863.977} C_VEL
LIN {X 0,Y 233.013,Z 522.807,A -85,B 0,C 180,E1 -19866.915,E2 -19866.915} C_VEL
LIN {X 0,Y 230.134,Z 530.64,A -85,B 0,C 180,E1 -19870.372,E2 -19870.372} C_VEL
LIN {X 0,Y 228.038,Z 536.879,A -85,B 0,C 180,E1 -19873.897,E2 -19873.897} C_VEL
LIN {X 0,Y 226.566,Z 541.708,A -85,B 0,C 180,E1 -19877.459,E2 -19877.459} C_VEL
LIN {X 0,Y 225.809,Z 545.254,A -85,B 0,C 180,E1 -19881.048,E2 -19881.048} C_VEL
LIN {X 0,Y 225.56,Z 547.592,A -85,B 0,C 180,E1 -19884.637,E2 -19884.637} C_VEL
LIN {X 0,Y 225.633,Z 548.77,A -85,B 0,C 180,E1 -19888.215,E2 -19888.215} C_VEL
LIN {X 0,Y 225.714,Z 548.927,A -85,B 0,C 180,E1 -19890,E2 -19890} C_VEL
LIN {X 0,Y 225.548,Z 548.31,A -85,B 0,C 180,E1 -19893.573,E2 -19893.573} C_VEL
LIN {X 0,Y 225.617,Z 546.539,A -85,B 0,C 180,E1 -19897.158,E2 -19897.158} C_VEL
LIN {X 0,Y 226.13,Z 543.592,A -85,B 0,C 180,E1 -19900.747,E2 -19900.747} C_VEL
LIN {X 0,Y 227.244,Z 539.406,A -85,B 0,C 180,E1 -19904.324,E2 -19904.324} C_VEL
LIN {X 0,Y 228.884,Z 533.865,A -85,B 0,C 180,E1 -19907.881,E2 -19907.881} C_VEL
LIN {X 0,Y 231.449,Z 526.832,A -85,B 0,C 180,E1 -19911.369,E2 -19911.369} C_VEL
LIN {X 0,Y 234.348,Z 519.317,A -85,B 0,C 180,E1 -19914.352,E2 -19914.352} C_VEL
LIN {X 0,Y 237.866,Z 509.747,A -85,B 0,C 180,E1 -19917.43,E2 -19917.43} C_VEL
LIN {X 0,Y 241.678,Z 499.379,A -85,B 0,C 180,E1 -19920.107,E2 -19920.107} C_VEL
LIN {X 0,Y 245.925,Z 487.152,A -85,B 0,C 180,E1 -19922.642,E2 -19922.642} C_VEL
LIN {X 0,Y 249.97,Z 474.69,A -85,B 0,C 180,E1 -19924.703,E2 -19924.703} C_VEL
LIN {X 0,Y 253.653,Z 461.605,A -85,B 0,C 180,E1 -19926.452,E2 -19926.452} C_VEL
LIN {X 0,Y 257.137,Z 447.349,A -85,B 0,C 180,E1 -19927.948,E2 -19927.948} C_VEL
LIN {X 0,Y 259.898,Z 433.553,A -85,B 0,C 180,E1 -19929.079,E2 -19929.079} C_VEL
LIN {X 0,Y 262.44,Z 418.107,A -85,B 0,C 180,E1 -19929.993,E2 -19929.993} C_VEL
LIN {X 0,Y 264.197,Z 402.816,A -85,B 0,C 180,E1 -19930.609,E2 -19930.609} C_VEL
LIN {X 0,Y 269.353,Z 307.667,A -85,B 0,C 180,E1 -19933.033,E2 -19933.033} C_VEL
LIN {X 0,Y 263.203,Z 293.254,A -85,B 0,C 180,E1 -19934.825,E2 -19934.825} C_VEL
LIN {X 0,Y 256.431,Z 279.457,A -85,B 0,C 180,E1 -19936.886,E2 -19936.886} C_VEL
LIN {X 0,Y 250.827,Z 269.379,A -85,B 0,C 180,E1 -19938.685,E2 -19938.685} C_VEL
LIN {X 0,Y 244.784,Z 259.268,A -85,B 0,C 180,E1 -19940.763,E2 -19940.763} C_VEL
LIN {X 0,Y 239.684,Z 251.17,A -85,B 0,C 180,E1 -19942.656,E2 -19942.656} C_VEL
LIN {X 0,Y 235.937,Z 245.695,A -85,B 0,C 180,E1 -19944.132,E2 -19944.132} C_VEL
LIN {X 0,Y 232.107,Z 240.322,A -85,B 0,C 180,E1 -19945.737,E2 -19945.737} C_VEL
LIN {X 0,Y 228.64,Z 236.074,A -85,B 0,C 180,E1 -19947.262,E2 -19947.262} C_VEL
LIN {X 0,Y 228.089,Z 234.584,A -85,B 0,C 180,E1 -19947.631,E2 -19947.631} C_VEL
LIN {X 0,Y 227.879,Z 233.717,A -85,B 0,C 180,E1 -19948.25,E2 -19948.25} C_VEL
LIN {X 0,Y 227.883,Z 233.717,A -85,B 0,C 180,E1 -19952.445,E2 -19952.445} C_VEL
LIN {X 0,Y 227.902,Z 233.7,A -85,B 0,C 180,E1 -19956.366,E2 -19956.366} C_VEL
LIN {X 0,Y 227.933,Z 233.695,A -85,B 0,C 180,E1 -19960.174,E2 -19960.174} C_VEL
LIN {X 0,Y 228.052,Z 233.694,A -85,B 0,C 180,E1 -19963.898,E2 -19963.898} C_VEL
LIN {X 0,Y 228.066,Z 233.691,A -85,B 0,C 180,E1 -19967.543,E2 -19967.543} C_VEL
LIN {X 0,Y 228.262,Z 233.667,A -85,B 0,C 180,E1 -19971.145,E2 -19971.145} C_VEL
LIN {X 0,Y 228.319,Z 233.666,A -85,B 0,C 180,E1 -19972.928,E2 -19972.928} C_VEL
LIN {X 0,Y 228.549,Z 233.641,A -85,B 0,C 180,E1 -19978.238,E2 -19978.238} C_VEL
LIN {X 0,Y 228.55,Z 233.64,A -85,B 0,C 180,E1 -19981.762,E2 -19981.762} C_VEL
LIN {X 0,Y 228.335,Z 233.666,A -85,B 0,C 180,E1 -19987.072,E2 -19987.072} C_VEL
LIN {X 0,Y 228.141,Z 233.692,A -85,B 0,C 180,E1 -19990.652,E2 -19990.652} C_VEL
LIN {X 0,Y 228.055,Z 233.701,A -85,B 0,C 180,E1 -19994.273,E2 -19994.273} C_VEL
LIN {X 0,Y 227.998,Z 233.705,A -85,B 0,C 180,E1 -19997.954,E2 -19997.954} C_VEL
LIN {X 0,Y 227.913,Z 233.721,A -85,B 0,C 180,E1 -20002.321,E2 -20002.321} C_VEL
LIN {X 0,Y 227.939,Z 233.68,A -85,B 0,C 180,E1 -20006.603,E2 -20006.603} C_VEL
LIN {X 0,Y 227.905,Z 233.716,A -85,B 0,C 180,E1 -20010.297,E2 -20010.297} C_VEL
LIN {X 0,Y 227.902,Z 233.729,A -85,B 0,C 180,E1 -20012.759,E2 -20012.759} C_VEL
LIN {X 0,Y 228.78,Z 236.348,A -85,B 0,C 180,E1 -20013.251,E2 -20013.251} C_VEL
LIN {X 0,Y 230.6,Z 238.481,A -85,B 0,C 180,E1 -20014.057,E2 -20014.057} C_VEL
LIN {X 0,Y 231.981,Z 239.441,A -85,B 0,C 180,E1 -20014.614,E2 -20014.614} C_VEL
LIN {X 0,Y 233.951,Z 242.712,A -85,B 0,C 180,E1 -20015.483,E2 -20015.483} C_VEL
LIN {X 0,Y 235.974,Z 244.788,A -85,B 0,C 180,E1 -20016.278,E2 -20016.278} C_VEL
LIN {X 0,Y 238.62,Z 248.449,A -85,B 0,C 180,E1 -20017.321,E2 -20017.321} C_VEL
LIN {X 0,Y 240.059,Z 250.362,A -85,B 0,C 180,E1 -20017.864,E2 -20017.864} C_VEL
LIN {X 0,Y 243.783,Z 255.405,A -85,B 0,C 180,E1 -20019.217,E2 -20019.217} C_VEL
LIN {X 0,Y 249.936,Z 264.189,A -85,B 0,C 180,E1 -20021.306,E2 -20021.306} C_VEL
LIN {X 0,Y 257.932,Z 276.506,A -85,B 0,C 180,E1 -20023.793,E2 -20023.793} C_VEL
LIN {X 0,Y 263.065,Z 285.609,A -85,B 0,C 180,E1 -20025.301,E2 -20025.301} C_VEL
LIN {X 0,Y 269.697,Z 299.905,A -85,B 0,C 180,E1 -20027.201,E2 -20027.201} C_VEL
LIN {X 0,Y 264.675,Z 391.792,A -85,B 0,C 180,E1 -20029.543,E2 -20029.543} C_VEL
LIN {X 0,Y 263.056,Z 406.935,A -85,B 0,C 180,E1 -20030.182,E2 -20030.182} C_VEL
LIN {X 0,Y 260.853,Z 421.664,A -85,B 0,C 180,E1 -20031.091,E2 -20031.091} C_VEL
LIN {X 0,Y 258.072,Z 436.177,A -85,B 0,C 180,E1 -20032.301,E2 -20032.301} C_VEL
LIN {X 0,Y 254.783,Z 450.572,A -85,B 0,C 180,E1 -20033.871,E2 -20033.871} C_VEL
LIN {X 0,Y 251.01,Z 464.019,A -85,B 0,C 180,E1 -20035.704,E2 -20035.704} C_VEL
LIN {X 0,Y 247.143,Z 476.222,A -85,B 0,C 180,E1 -20037.779,E2 -20037.779} C_VEL
LIN {X 0,Y 243.315,Z 487.129,A -85,B 0,C 180,E1 -20040.058,E2 -20040.058} C_VEL
LIN {X 0,Y 239.916,Z 496.677,A -85,B 0,C 180,E1 -20042.525,E2 -20042.525} C_VEL
LIN {X 0,Y 236.339,Z 505.863,A -85,B 0,C 180,E1 -20045.398,E2 -20045.398} C_VEL
LIN {X 0,Y 233.297,Z 513.495,A -85,B 0,C 180,E1 -20048.345,E2 -20048.345} C_VEL
LIN {X 0,Y 230.838,Z 519.822,A -85,B 0,C 180,E1 -20051.357,E2 -20051.357} C_VEL
LIN {X 0,Y 228.714,Z 525.628,A -85,B 0,C 180,E1 -20054.86,E2 -20054.86} C_VEL
LIN {X 0,Y 227.528,Z 529.064,A -85,B 0,C 180,E1 -20057.513,E2 -20057.513} C_VEL
LIN {X 0,Y 226.511,Z 532.538,A -85,B 0,C 180,E1 -20061.076,E2 -20061.076} C_VEL
LIN {X 0,Y 225.923,Z 534.832,A -85,B 0,C 180,E1 -20064.645,E2 -20064.645} C_VEL
LIN {X 0,Y 225.738,Z 535.998,A -85,B 0,C 180,E1 -20068.216,E2 -20068.216} C_VEL
LIN {X 0,Y 225.737,Z 536.01,A -85,B 0,C 180,E1 -20071.784,E2 -20071.784} C_VEL
LIN {X 0,Y 225.916,Z 534.855,A -85,B 0,C 180,E1 -20075.445,E2 -20075.445} C_VEL
LIN {X 0,Y 226.462,Z 532.651,A -85,B 0,C 180,E1 -20078.926,E2 -20078.926} C_VEL
LIN {X 0,Y 227.493,Z 529.22,A -85,B 0,C 180,E1 -20082.489,E2 -20082.489} C_VEL
LIN {X 0,Y 229.203,Z 524.517,A -85,B 0,C 180,E1 -20086.019,E2 -20086.019} C_VEL
LIN {X 0,Y 231.499,Z 518.421,A -85,B 0,C 180,E1 -20089.508,E2 -20089.508} C_VEL
LIN {X 0,Y 234.475,Z 510.74,A -85,B 0,C 180,E1 -20092.932,E2 -20092.932} C_VEL
LIN {X 0,Y 237.716,Z 502.546,A -85,B 0,C 180,E1 -20095.853,E2 -20095.853} C_VEL
LIN {X 0,Y 241.497,Z 492.668,A -85,B 0,C 180,E1 -20098.696,E2 -20098.696} C_VEL
LIN {X 0,Y 245.048,Z 482.541,A -85,B 0,C 180,E1 -20101.08,E2 -20101.08} C_VEL
LIN {X 0,Y 249.115,Z 470.472,A -85,B 0,C 180,E1 -20103.375,E2 -20103.375} C_VEL
LIN {X 0,Y 252.701,Z 458.367,A -85,B 0,C 180,E1 -20105.245,E2 -20105.245} C_VEL
LIN {X 0,Y 256.171,Z 445.206,A -85,B 0,C 180,E1 -20106.879,E2 -20106.879} C_VEL
LIN {X 0,Y 259.162,Z 431.442,A -85,B 0,C 180,E1 -20108.243,E2 -20108.243} C_VEL
LIN {X 0,Y 261.77,Z 416.658,A -85,B 0,C 180,E1 -20109.366,E2 -20109.366} C_VEL
LIN {X 0,Y 263.651,Z 402.649,A -85,B 0,C 180,E1 -20110.146,E2 -20110.146} C_VEL
LIN {X 0,Y 265.102,Z 387.827,A -85,B 0,C 180,E1 -20110.691,E2 -20110.691} C_VEL
LIN {X 0,Y 269.231,Z 309.941,A -85,B 0,C 180,E1 -20112.678,E2 -20112.678} C_VEL
LIN {X 0,Y 269.749,Z 299.865,A -85,B 0,C 180,E1 -20112.935,E2 -20112.935} C_VEL
LIN {X 0,Y 263.175,Z 285.712,A -85,B 0,C 180,E1 -20114.822,E2 -20114.822} C_VEL
LIN {X 0,Y 258.832,Z 277.946,A -85,B 0,C 180,E1 -20116.096,E2 -20116.096} C_VEL
LIN {X 0,Y 250.475,Z 264.905,A -85,B 0,C 180,E1 -20118.686,E2 -20118.686} C_VEL
LIN {X 0,Y 244.266,Z 256.029,A -85,B 0,C 180,E1 -20120.787,E2 -20120.787} C_VEL
LIN {X 0,Y 241.676,Z 252.528,A -85,B 0,C 180,E1 -20121.715,E2 -20121.715} C_VEL
LIN {X 0,Y 238.748,Z 248.523,A -85,B 0,C 180,E1 -20122.816,E2 -20122.816} C_VEL
LIN {X 0,Y 236.07,Z 244.871,A -85,B 0,C 180,E1 -20123.872,E2 -20123.872} C_VEL
LIN {X 0,Y 232.806,Z 241.049,A -85,B 0,C 180,E1 -20125.198,E2 -20125.198} C_VEL
LIN {X 0,Y 231.873,Z 239.235,A -85,B 0,C 180,E1 -20125.631,E2 -20125.631} C_VEL
LIN {X 0,Y 229.412,Z 237.281,A -85,B 0,C 180,E1 -20126.656,E2 -20126.656} C_VEL
LIN {X 0,Y 228.197,Z 234.997,A -85,B 0,C 180,E1 -20127.256,E2 -20127.256} C_VEL
LIN {X 0,Y 227.917,Z 233.688,A -85,B 0,C 180,E1 -20127.473,E2 -20127.473} C_VEL
LIN {X 0,Y 227.916,Z 233.698,A -85,B 0,C 180,E1 -20130.437,E2 -20130.437} C_VEL
LIN {X 0,Y 227.925,Z 233.711,A -85,B 0,C 180,E1 -20134.425,E2 -20134.425} C_VEL
LIN {X 0,Y 227.958,Z 233.707,A -85,B 0,C 180,E1 -20138.286,E2 -20138.286} C_VEL
LIN {X 0,Y 228.031,Z 233.701,A -85,B 0,C 180,E1 -20142.826,E2 -20142.826} C_VEL
LIN {X 0,Y 228.088,Z 233.698,A -85,B 0,C 180,E1 -20147.544,E2 -20147.544} C_VEL
LIN {X 0,Y 228.3,Z 233.662,A -85,B 0,C 180,E1 -20151.146,E2 -20151.146} C_VEL
LIN {X 0,Y 228.348,Z 233.665,A -85,B 0,C 180,E1 -20152.928,E2 -20152.928} C_VEL
LIN {X 0,Y 228.549,Z 233.633,A -85,B 0,C 180,E1 -20158.238,E2 -20158.238} C_VEL
LIN {X 0,Y 228.549,Z 233.642,A -85,B 0,C 180,E1 -20161.762,E2 -20161.762} C_VEL
LIN {X 0,Y 228.434,Z 233.649,A -85,B 0,C 180,E1 -20162.302,E2 -20162.302} C_VEL
LIN {X 0,Y 227.588,Z 233.75,A -85,B 0,C 180,E1 -20163.772,E2 -20163.772} C_VEL
LIN {X 0,Y 224.714,Z 234.12,A -85,B 0,C 180,E1 -20166.175,E2 -20166.175} C_VEL
LIN {X 0,Y 221.519,Z 234.512,A -85,B 0,C 180,E1 -20169.14,E2 -20169.14} C_VEL
LIN {X 0,Y 221.14,Z 234.56,A -85,B 0,C 180,E1 -20170.166,E2 -20170.166} C_VEL
LIN {X 0,Y 220.987,Z 234.584,A -85,B 0,C 180,E1 -20174.739,E2 -20174.739} C_VEL
LIN {X 0,Y 220.917,Z 234.587,A -85,B 0,C 180,E1 -20178.55,E2 -20178.55} C_VEL
LIN {X 0,Y 220.892,Z 234.591,A -85,B 0,C 180,E1 -20182.683,E2 -20182.683} C_VEL
LIN {X 0,Y 220.882,Z 234.595,A -85,B 0,C 180,E1 -20187.016,E2 -20187.016} C_VEL
LIN {X 0,Y 220.853,Z 234.602,A -85,B 0,C 180,E1 -20189.227,E2 -20189.227} C_VEL
LIN {X 0,Y 221.826,Z 237.386,A -85,B 0,C 180,E1 -20189.868,E2 -20189.868} C_VEL
LIN {X 0,Y 223.881,Z 239.593,A -85,B 0,C 180,E1 -20190.9,E2 -20190.9} C_VEL
LIN {X 0,Y 225.212,Z 240.545,A -85,B 0,C 180,E1 -20191.514,E2 -20191.514} C_VEL
LIN {X 0,Y 227.158,Z 243.745,A -85,B 0,C 180,E1 -20192.484,E2 -20192.484} C_VEL
LIN {X 0,Y 230.466,Z 247.752,A -85,B 0,C 180,E1 -20193.964,E2 -20193.964} C_VEL
LIN {X 0,Y 233.511,Z 252.137,A -85,B 0,C 180,E1 -20195.279,E2 -20195.279} C_VEL
LIN {X 0,Y 238.594,Z 260.046,A -85,B 0,C 180,E1 -20197.343,E2 -20197.343} C_VEL
LIN {X 0,Y 246.1,Z 272.453,A -85,B 0,C 180,E1 -20200.115,E2 -20200.115} C_VEL
LIN {X 0,Y 253.17,Z 285.547,A -85,B 0,C 180,E1 -20202.507,E2 -20202.507} C_VEL
LIN {X 0,Y 259.698,Z 299.395,A -85,B 0,C 180,E1 -20204.582,E2 -20204.582} C_VEL
LIN {X 0,Y 264.111,Z 309.894,A -85,B 0,C 180,E1 -20205.928,E2 -20205.928} C_VEL
LIN {X 0,Y 260.807,Z 371.513,A -85,B 0,C 180,E1 -20207.515,E2 -20207.515} C_VEL
LIN {X 0,Y 258.819,Z 403.614,A -85,B 0,C 180,E1 -20208.363,E2 -20208.363} C_VEL
LIN {X 0,Y 257.002,Z 419.339,A -85,B 0,C 180,E1 -20209.047,E2 -20209.047} C_VEL
LIN {X 0,Y 254.488,Z 433.828,A -85,B 0,C 180,E1 -20209.925,E2 -20209.925} C_VEL
LIN {X 0,Y 251.574,Z 447.568,A -85,B 0,C 180,E1 -20211.057,E2 -20211.057} C_VEL
LIN {X 0,Y 247.963,Z 461.971,A -85,B 0,C 180,E1 -20212.612,E2 -20212.612} C_VEL
LIN {X 0,Y 244.157,Z 474.746,A -85,B 0,C 180,E1 -20214.347,E2 -20214.347} C_VEL
LIN {X 0,Y 239.933,Z 487.165,A -85,B 0,C 180,E1 -20216.436,E2 -20216.436} C_VEL
LIN {X 0,Y 235.529,Z 499.348,A -85,B 0,C 180,E1 -20219.022,E2 -20219.022} C_VEL
LIN {X 0,Y 231.739,Z 509.092,A -85,B 0,C 180,E1 -20221.58,E2 -20221.58} C_VEL
LIN {X 0,Y 228.358,Z 518.017,A -85,B 0,C 180,E1 -20224.478,E2 -20224.478} C_VEL
LIN {X 0,Y 225.197,Z 525.72,A -85,B 0,C 180,E1 -20227.524,E2 -20227.524} C_VEL
LIN {X 0,Y 222.768,Z 532.116,A -85,B 0,C 180,E1 -20230.655,E2 -20230.655} C_VEL
LIN {X 0,Y 220.704,Z 538.003,A -85,B 0,C 180,E1 -20234.296,E2 -20234.296} C_VEL
LIN {X 0,Y 219.583,Z 541.506,A -85,B 0,C 180,E1 -20237.054,E2 -20237.054} C_VEL
LIN {X 0,Y 218.754,Z 545.053,A -85,B 0,C 180,E1 -20240.756,E2 -20240.756} C_VEL
LIN {X 0,Y 218.476,Z 547.391,A -85,B 0,C 180,E1 -20244.462,E2 -20244.462} C_VEL
LIN {X 0,Y 218.529,Z 548.569,A -85,B 0,C 180,E1 -20248.157,E2 -20248.157} C_VEL
LIN {X 0,Y 218.628,Z 548.726,A -85,B 0,C 180,E1 -20250,E2 -20250} C_VEL
LIN {X 0,Y 218.449,Z 548.108,A -85,B 0,C 180,E1 -20253.689,E2 -20253.689} C_VEL
LIN {X 0,Y 218.552,Z 546.337,A -85,B 0,C 180,E1 -20257.39,E2 -20257.39} C_VEL
LIN {X 0,Y 219.111,Z 543.389,A -85,B 0,C 180,E1 -20261.096,E2 -20261.096} C_VEL
LIN {X 0,Y 220.313,Z 539.202,A -85,B 0,C 180,E1 -20264.785,E2 -20264.785} C_VEL
LIN {X 0,Y 222.095,Z 533.661,A -85,B 0,C 180,E1 -20268.447,E2 -20268.447} C_VEL
LIN {X 0,Y 224.798,Z 526.628,A -85,B 0,C 180,E1 -20272.034,E2 -20272.034} C_VEL
LIN {X 0,Y 227.863,Z 519.113,A -85,B 0,C 180,E1 -20275.093,E2 -20275.093} C_VEL
LIN {X 0,Y 231.258,Z 510.199,A -85,B 0,C 180,E1 -20278.049,E2 -20278.049} C_VEL
LIN {X 0,Y 235.507,Z 499.174,A -85,B 0,C 180,E1 -20280.982,E2 -20280.982} C_VEL
LIN {X 0,Y 239.932,Z 486.946,A -85,B 0,C 180,E1 -20283.564,E2 -20283.564} C_VEL
LIN {X 0,Y 244.144,Z 474.485,A -85,B 0,C 180,E1 -20285.655,E2 -20285.655} C_VEL
LIN {X 0,Y 247.699,Z 462.301,A -85,B 0,C 180,E1 -20287.321,E2 -20287.321} C_VEL
LIN {X 0,Y 251.118,Z 448.979,A -85,B 0,C 180,E1 -20288.77,E2 -20288.77} C_VEL
LIN {X 0,Y 254.185,Z 434.481,A -85,B 0,C 180,E1 -20290.003,E2 -20290.003} C_VEL
LIN {X 0,Y 256.786,Z 419.459,A -85,B 0,C 180,E1 -20290.93,E2 -20290.93} C_VEL
LIN {X 0,Y 258.736,Z 403.775,A -85,B 0,C 180,E1 -20291.588,E2 -20291.588} C_VEL
LIN {X 0,Y 261.191,Z 362.226,A -85,B 0,C 180,E1 -20292.69,E2 -20292.69} C_VEL
LIN {X 0,Y 263.988,Z 309.762,A -85,B 0,C 180,E1 -20294.044,E2 -20294.044} C_VEL
LIN {X 0,Y 258.521,Z 296.852,A -85,B 0,C 180,E1 -20295.718,E2 -20295.718} C_VEL
LIN {X 0,Y 252.291,Z 283.913,A -85,B 0,C 180,E1 -20297.708,E2 -20297.708} C_VEL
LIN {X 0,Y 245.458,Z 271.457,A -85,B 0,C 180,E1 -20300.027,E2 -20300.027} C_VEL
LIN {X 0,Y 238.795,Z 260.424,A -85,B 0,C 180,E1 -20302.487,E2 -20302.487} C_VEL
LIN {X 0,Y 236.025,Z 256.078,A -85,B 0,C 180,E1 -20303.581,E2 -20303.581} C_VEL
LIN {X 0,Y 232.767,Z 251.206,A -85,B 0,C 180,E1 -20304.927,E2 -20304.927} C_VEL
LIN {X 0,Y 229.29,Z 246.202,A -85,B 0,C 180,E1 -20306.449,E2 -20306.449} C_VEL
LIN {X 0,Y 225.799,Z 241.805,A -85,B 0,C 180,E1 -20308.054,E2 -20308.054} C_VEL
LIN {X 0,Y 225.034,Z 240.224,A -85,B 0,C 180,E1 -20308.459,E2 -20308.459} C_VEL
LIN {X 0,Y 222.605,Z 238.443,A -85,B 0,C 180,E1 -20309.594,E2 -20309.594} C_VEL
LIN {X 0,Y 221.291,Z 236.23,A -85,B 0,C 180,E1 -20310.314,E2 -20310.314} C_VEL
LIN {X 0,Y 220.874,Z 234.587,A -85,B 0,C 180,E1 -20310.646,E2 -20310.646} C_VEL
LIN {X 0,Y 220.891,Z 234.586,A -85,B 0,C 180,E1 -20313.549,E2 -20313.549} C_VEL
LIN {X 0,Y 220.86,Z 234.562,A -85,B 0,C 180,E1 -20317.552,E2 -20317.552} C_VEL
LIN {X 0,Y 220.98,Z 234.58,A -85,B 0,C 180,E1 -20322.571,E2 -20322.571} C_VEL
LIN {X 0,Y 221.006,Z 234.571,A -85,B 0,C 180,E1 -20327.138,E2 -20327.138} C_VEL
LIN {X 0,Y 221.2,Z 234.548,A -85,B 0,C 180,E1 -20330.859,E2 -20330.859} C_VEL
LIN {X 0,Y 221.254,Z 234.543,A -85,B 0,C 180,E1 -20332.701,E2 -20332.701} C_VEL
LIN {X 0,Y 221.507,Z 234.518,A -85,B 0,C 180,E1 -20338.182,E2 -20338.182} C_VEL
LIN {X 0,Y 221.507,Z 234.517,A -85,B 0,C 180,E1 -20341.818,E2 -20341.818} C_VEL
LIN {X 0,Y 221.267,Z 234.544,A -85,B 0,C 180,E1 -20347.299,E2 -20347.299} C_VEL
LIN {X 0,Y 221.077,Z 234.573,A -85,B 0,C 180,E1 -20350.996,E2 -20350.996} C_VEL
LIN {X 0,Y 221.01,Z 234.57,A -85,B 0,C 180,E1 -20356.631,E2 -20356.631} C_VEL
LIN {X 0,Y 220.88,Z 234.587,A -85,B 0,C 180,E1 -20360.488,E2 -20360.488} C_VEL
LIN {X 0,Y 220.858,Z 234.571,A -85,B 0,C 180,E1 -20364.436,E2 -20364.436} C_VEL
LIN {X 0,Y 220.833,Z 234.589,A -85,B 0,C 180,E1 -20368.514,E2 -20368.514} C_VEL
LIN {X 0,Y 220.878,Z 234.595,A -85,B 0,C 180,E1 -20369.813,E2 -20369.813} C_VEL
LIN {X 0,Y 221.668,Z 237.077,A -85,B 0,C 180,E1 -20370.351,E2 -20370.351} C_VEL
LIN {X 0,Y 223.45,Z 239.254,A -85,B 0,C 180,E1 -20371.263,E2 -20371.263} C_VEL
LIN {X 0,Y 225.155,Z 240.473,A -85,B 0,C 180,E1 -20372.049,E2 -20372.049} C_VEL
LIN {X 0,Y 227.011,Z 243.604,A -85,B 0,C 180,E1 -20372.975,E2 -20372.975} C_VEL
LIN {X 0,Y 229.255,Z 245.711,A -85,B 0,C 180,E1 -20373.954,E2 -20373.954} C_VEL
LIN {X 0,Y 231.559,Z 249.069,A -85,B 0,C 180,E1 -20374.978,E2 -20374.978} C_VEL
LIN {X 0,Y 233.281,Z 251.056,A -85,B 0,C 180,E1 -20375.686,E2 -20375.686} C_VEL
LIN {X 0,Y 237.116,Z 256.313,A -85,B 0,C 180,E1 -20377.227,E2 -20377.227} C_VEL
LIN {X 0,Y 242.797,Z 264.169,A -85,B 0,C 180,E1 -20379.333,E2 -20379.333} C_VEL
LIN {X 0,Y 250.122,Z 275.161,A -85,B 0,C 180,E1 -20381.821,E2 -20381.821} C_VEL
LIN {X 0,Y 257.464,Z 287.37,A -85,B 0,C 180,E1 -20384.113,E2 -20384.113} C_VEL
LIN {X 0,Y 263.351,Z 299.864,A -85,B 0,C 180,E1 -20385.897,E2 -20385.897} C_VEL
LIN {X 0,Y 264.406,Z 302.208,A -85,B 0,C 180,E1 -20386.207,E2 -20386.207} C_VEL
LIN {X 0,Y 259.329,Z 392.008,A -85,B 0,C 180,E1 -20388.528,E2 -20388.528} C_VEL
LIN {X 0,Y 257.531,Z 407.923,A -85,B 0,C 180,E1 -20389.214,E2 -20389.214} C_VEL
LIN {X 0,Y 255.165,Z 423.034,A -85,B 0,C 180,E1 -20390.181,E2 -20390.181} C_VEL
LIN {X 0,Y 252.35,Z 437.052,A -85,B 0,C 180,E1 -20391.382,E2 -20391.382} C_VEL
LIN {X 0,Y 249.09,Z 450.778,A -85,B 0,C 180,E1 -20392.909,E2 -20392.909} C_VEL
LIN {X 0,Y 245.179,Z 464.224,A -85,B 0,C 180,E1 -20394.77,E2 -20394.77} C_VEL
LIN {X 0,Y 241.173,Z 476.426,A -85,B 0,C 180,E1 -20396.881,E2 -20396.881} C_VEL
LIN {X 0,Y 236.952,Z 487.897,A -85,B 0,C 180,E1 -20399.333,E2 -20399.333} C_VEL
LIN {X 0,Y 233.641,Z 496.88,A -85,B 0,C 180,E1 -20401.722,E2 -20401.722} C_VEL
LIN {X 0,Y 229.861,Z 506.067,A -85,B 0,C 180,E1 -20404.657,E2 -20404.657} C_VEL
LIN {X 0,Y 226.671,Z 513.699,A -85,B 0,C 180,E1 -20407.678,E2 -20407.678} C_VEL
LIN {X 0,Y 224.083,Z 520.025,A -85,B 0,C 180,E1 -20410.773,E2 -20410.773} C_VEL
LIN {X 0,Y 221.83,Z 525.831,A -85,B 0,C 180,E1 -20414.378,E2 -20414.378} C_VEL
LIN {X 0,Y 220.566,Z 529.267,A -85,B 0,C 180,E1 -20417.112,E2 -20417.112} C_VEL
LIN {X 0,Y 219.473,Z 532.74,A -85,B 0,C 180,E1 -20420.787,E2 -20420.787} C_VEL
LIN {X 0,Y 218.838,Z 535.09,A -85,B 0,C 180,E1 -20424.606,E2 -20424.606} C_VEL
LIN {X 0,Y 218.656,Z 536.198,A -85,B 0,C 180,E1 -20428.158,E2 -20428.158} C_VEL
LIN {X 0,Y 218.656,Z 536.211,A -85,B 0,C 180,E1 -20431.842,E2 -20431.842} C_VEL
LIN {X 0,Y 218.847,Z 535.095,A -85,B 0,C 180,E1 -20435.528,E2 -20435.528} C_VEL
LIN {X 0,Y 219.434,Z 532.851,A -85,B 0,C 180,E1 -20439.215,E2 -20439.215} C_VEL
LIN {X 0,Y 220.539,Z 529.421,A -85,B 0,C 180,E1 -20442.889,E2 -20442.889} C_VEL
LIN {X 0,Y 222.369,Z 524.717,A -85,B 0,C 180,E1 -20446.525,E2 -20446.525} C_VEL
LIN {X 0,Y 224.789,Z 518.621,A -85,B 0,C 180,E1 -20450.115,E2 -20450.115} C_VEL
LIN {X 0,Y 227.473,Z 511.996,A -85,B 0,C 180,E1 -20453.198,E2 -20453.198} C_VEL
LIN {X 0,Y 230.816,Z 503.978,A -85,B 0,C 180,E1 -20456.199,E2 -20456.199} C_VEL
LIN {X 0,Y 234.68,Z 494.426,A -85,B 0,C 180,E1 -20459.095,E2 -20459.095} C_VEL
LIN {X 0,Y 238.293,Z 484.516,A -85,B 0,C 180,E1 -20461.566,E2 -20461.566} C_VEL
LIN {X 0,Y 242.516,Z 472.798,A -85,B 0,C 180,E1 -20463.907,E2 -20463.907} C_VEL
LIN {X 0,Y 245.762,Z 462.422,A -85,B 0,C 180,E1 -20465.637,E2 -20465.637} C_VEL
LIN {X 0,Y 249.381,Z 450.128,A -85,B 0,C 180,E1 -20467.293,E2 -20467.293} C_VEL
LIN {X 0,Y 252.496,Z 436.987,A -85,B 0,C 180,E1 -20468.746,E2 -20468.746} C_VEL
LIN {X 0,Y 255.487,Z 422.026,A -85,B 0,C 180,E1 -20470.015,E2 -20470.015} C_VEL
LIN {X 0,Y 257.838,Z 406.492,A -85,B 0,C 180,E1 -20470.985,E2 -20470.985} C_VEL
LIN {X 0,Y 259.525,Z 391.014,A -85,B 0,C 180,E1 -20471.628,E2 -20471.628} C_VEL
LIN {X 0,Y 264.021,Z 311.157,A -85,B 0,C 180,E1 -20473.691,E2 -20473.691} C_VEL
LIN {X 0,Y 264.467,Z 302.216,A -85,B 0,C 180,E1 -20473.928,E2 -20473.928} C_VEL
LIN {X 0,Y 258.071,Z 288.382,A -85,B 0,C 180,E1 -20475.862,E2 -20475.862} C_VEL
LIN {X 0,Y 251.411,Z 277.16,A -85,B 0,C 180,E1 -20477.927,E2 -20477.927} C_VEL
LIN {X 0,Y 243.962,Z 265.79,A -85,B 0,C 180,E1 -20480.43,E2 -20480.43} C_VEL
LIN {X 0,Y 238.653,Z 258.374,A -85,B 0,C 180,E1 -20482.366,E2 -20482.366} C_VEL
LIN {X 0,Y 235.286,Z 253.789,A -85,B 0,C 180,E1 -20483.681,E2 -20483.681} C_VEL
LIN {X 0,Y 232.302,Z 249.79,A -85,B 0,C 180,E1 -20484.913,E2 -20484.913} C_VEL
LIN {X 0,Y 229.671,Z 246.408,A -85,B 0,C 180,E1 -20486.051,E2 -20486.051} C_VEL
LIN {X 0,Y 228.817,Z 245.248,A -85,B 0,C 180,E1 -20486.436,E2 -20486.436} C_VEL
LIN {X 0,Y 226.328,Z 242.658,A -85,B 0,C 180,E1 -20487.555,E2 -20487.555} C_VEL
LIN {X 0,Y 224.868,Z 240.121,A -85,B 0,C 180,E1 -20488.301,E2 -20488.301} C_VEL
LIN {X 0,Y 222.464,Z 238.27,A -85,B 0,C 180,E1 -20489.441,E2 -20489.441} C_VEL
LIN {X 0,Y 221.174,Z 235.932,A -85,B 0,C 180,E1 -20490.166,E2 -20490.166} C_VEL
LIN {X 0,Y 220.886,Z 234.573,A -85,B 0,C 180,E1 -20490.451,E2 -20490.451} C_VEL
LIN {X 0,Y 220.892,Z 234.585,A -85,B 0,C 180,E1 -20493.549,E2 -20493.549} C_VEL
LIN {X 0,Y 220.874,Z 234.586,A -85,B 0,C 180,E1 -20497.553,E2 -20497.553} C_VEL
LIN {X 0,Y 220.98,Z 234.576,A -85,B 0,C 180,E1 -20502.571,E2 -20502.571} C_VEL
LIN {X 0,Y 221.02,Z 234.573,A -85,B 0,C 180,E1 -20507.139,E2 -20507.139} C_VEL
LIN {X 0,Y 221.231,Z 234.54,A -85,B 0,C 180,E1 -20510.86,E2 -20510.86} C_VEL
LIN {X 0,Y 221.3,Z 234.545,A -85,B 0,C 180,E1 -20512.702,E2 -20512.702} C_VEL
LIN {X 0,Y 221.507,Z 234.51,A -85,B 0,C 180,E1 -20518.182,E2 -20518.182} C_VEL
LIN {X 0,Y 221.507,Z 234.519,A -85,B 0,C 180,E1 -20521.818,E2 -20521.818} C_VEL
LIN {X 0,Y 221.254,Z 234.544,A -85,B 0,C 180,E1 -20527.299,E2 -20527.299} C_VEL
LIN {X 0,Y 221.14,Z 234.56,A -85,B 0,C 180,E1 -20530.166,E2 -20530.166} C_VEL
LIN {X 0,Y 220.369,Z 234.661,A -85,B 0,C 180,E1 -20531.684,E2 -20531.684} C_VEL
LIN {X 0,Y 217.476,Z 235.015,A -85,B 0,C 180,E1 -20534.164,E2 -20534.164} C_VEL
LIN {X 0,Y 214.234,Z 235.416,A -85,B 0,C 180,E1 -20537.229,E2 -20537.229} C_VEL
LIN {X 0,Y 213.885,Z 235.461,A -85,B 0,C 180,E1 -20538.291,E2 -20538.291} C_VEL
LIN {X 0,Y 213.843,Z 235.474,A -85,B 0,C 180,E1 -20543.227,E2 -20543.227} C_VEL
LIN {X 0,Y 213.86,Z 235.651,A -85,B 0,C 180,E1 -20545.812,E2 -20545.812} C_VEL
LIN {X 0,Y 214.589,Z 237.854,A -85,B 0,C 180,E1 -20546.371,E2 -20546.371} C_VEL
LIN {X 0,Y 216.345,Z 240.082,A -85,B 0,C 180,E1 -20547.444,E2 -20547.444} C_VEL
LIN {X 0,Y 218.377,Z 241.42,A -85,B 0,C 180,E1 -20548.536,E2 -20548.536} C_VEL
LIN {X 0,Y 220.087,Z 244.424,A -85,B 0,C 180,E1 -20549.533,E2 -20549.533} C_VEL
LIN {X 0,Y 222.852,Z 247.15,A -85,B 0,C 180,E1 -20550.923,E2 -20550.923} C_VEL
LIN {X 0,Y 225.222,Z 250.503,A -85,B 0,C 180,E1 -20552.105,E2 -20552.105} C_VEL
LIN {X 0,Y 227.808,Z 253.93,A -85,B 0,C 180,E1 -20553.313,E2 -20553.313} C_VEL
LIN {X 0,Y 232.037,Z 260.406,A -85,B 0,C 180,E1 -20555.2,E2 -20555.2} C_VEL
LIN {X 0,Y 235.292,Z 265.423,A -85,B 0,C 180,E1 -20556.553,E2 -20556.553} C_VEL
LIN {X 0,Y 242.39,Z 277.436,A -85,B 0,C 180,E1 -20559.298,E2 -20559.298} C_VEL
LIN {X 0,Y 248.839,Z 289.559,A -85,B 0,C 180,E1 -20561.585,E2 -20561.585} C_VEL
LIN {X 0,Y 255.341,Z 303.55,A -85,B 0,C 180,E1 -20563.752,E2 -20563.752} C_VEL
LIN {X 0,Y 258.97,Z 312.361,A -85,B 0,C 180,E1 -20564.918,E2 -20564.918} C_VEL
LIN {X 0,Y 253.818,Z 400.748,A -85,B 0,C 180,E1 -20567.216,E2 -20567.216} C_VEL
LIN {X 0,Y 252.123,Z 415.744,A -85,B 0,C 180,E1 -20567.809,E2 -20567.809} C_VEL
LIN {X 0,Y 249.595,Z 431.136,A -85,B 0,C 180,E1 -20568.706,E2 -20568.706} C_VEL
LIN {X 0,Y 246.512,Z 445.387,A -85,B 0,C 180,E1 -20569.833,E2 -20569.833} C_VEL
LIN {X 0,Y 242.91,Z 459.593,A -85,B 0,C 180,E1 -20571.327,E2 -20571.327} C_VEL
LIN {X 0,Y 239.214,Z 471.96,A -85,B 0,C 180,E1 -20572.968,E2 -20572.968} C_VEL
LIN {X 0,Y 234.785,Z 484.82,A -85,B 0,C 180,E1 -20575.077,E2 -20575.077} C_VEL
LIN {X 0,Y 230.802,Z 495.594,A -85,B 0,C 180,E1 -20577.284,E2 -20577.284} C_VEL
LIN {X 0,Y 226.852,Z 505.568,A -85,B 0,C 180,E1 -20579.773,E2 -20579.773} C_VEL
LIN {X 0,Y 223.434,Z 514.077,A -85,B 0,C 180,E1 -20582.358,E2 -20582.358} C_VEL
LIN {X 0,Y 219.881,Z 522.405,A -85,B 0,C 180,E1 -20585.449,E2 -20585.449} C_VEL
LIN {X 0,Y 216.661,Z 530.236,A -85,B 0,C 180,E1 -20589.096,E2 -20589.096} C_VEL
LIN {X 0,Y 214.312,Z 536.475,A -85,B 0,C 180,E1 -20592.834,E2 -20592.834} C_VEL
LIN {X 0,Y 212.621,Z 541.305,A -85,B 0,C 180,E1 -20596.622,E2 -20596.622} C_VEL
LIN {X 0,Y 211.718,Z 544.852,A -85,B 0,C 180,E1 -20600.446,E2 -20600.446} C_VEL
LIN {X 0,Y 211.375,Z 547.189,A -85,B 0,C 180,E1 -20604.276,E2 -20604.276} C_VEL
LIN {X 0,Y 211.428,Z 548.368,A -85,B 0,C 180,E1 -20608.095,E2 -20608.095} C_VEL
LIN {X 0,Y 211.544,Z 548.526,A -85,B 0,C 180,E1 -20610,E2 -20610} C_VEL
LIN {X 0,Y 211.356,Z 547.857,A -85,B 0,C 180,E1 -20614.006,E2 -20614.006} C_VEL
LIN {X 0,Y 211.482,Z 546.135,A -85,B 0,C 180,E1 -20617.639,E2 -20617.639} C_VEL
LIN {X 0,Y 212.089,Z 543.186,A -85,B 0,C 180,E1 -20621.468,E2 -20621.468} C_VEL
LIN {X 0,Y 213.376,Z 538.998,A -85,B 0,C 180,E1 -20625.277,E2 -20625.277} C_VEL
LIN {X 0,Y 215.294,Z 533.457,A -85,B 0,C 180,E1 -20629.052,E2 -20629.052} C_VEL
LIN {X 0,Y 218.159,Z 526.423,A -85,B 0,C 180,E1 -20632.741,E2 -20632.741} C_VEL
LIN {X 0,Y 221.402,Z 518.909,A -85,B 0,C 180,E1 -20635.878,E2 -20635.878} C_VEL
LIN {X 0,Y 225.167,Z 509.449,A -85,B 0,C 180,E1 -20639.08,E2 -20639.08} C_VEL
LIN {X 0,Y 229.414,Z 498.969,A -85,B 0,C 180,E1 -20641.9,E2 -20641.9} C_VEL
LIN {X 0,Y 233.984,Z 486.74,A -85,B 0,C 180,E1 -20644.536,E2 -20644.536} C_VEL
LIN {X 0,Y 238.378,Z 474.279,A -85,B 0,C 180,E1 -20646.656,E2 -20646.656} C_VEL
LIN {X 0,Y 242.386,Z 461.006,A -85,B 0,C 180,E1 -20648.476,E2 -20648.476} C_VEL
LIN {X 0,Y 246.056,Z 446.934,A -85,B 0,C 180,E1 -20649.989,E2 -20649.989} C_VEL
LIN {X 0,Y 249.034,Z 433.137,A -85,B 0,C 180,E1 -20651.139,E2 -20651.139} C_VEL
LIN {X 0,Y 251.742,Z 417.685,A -85,B 0,C 180,E1 -20652.067,E2 -20652.067} C_VEL
LIN {X 0,Y 253.589,Z 402.383,A -85,B 0,C 180,E1 -20652.697,E2 -20652.697} C_VEL
LIN {X 0,Y 258.835,Z 312.174,A -85,B 0,C 180,E1 -20655.057,E2 -20655.057} C_VEL
LIN {X 0,Y 253.224,Z 298.83,A -85,B 0,C 180,E1 -20656.871,E2 -20656.871} C_VEL
LIN {X 0,Y 246.218,Z 284.514,A -85,B 0,C 180,E1 -20659.247,E2 -20659.247} C_VEL
LIN {X 0,Y 239.267,Z 272.12,A -85,B 0,C 180,E1 -20661.784,E2 -20661.784} C_VEL
LIN {X 0,Y 233.165,Z 262.015,A -85,B 0,C 180,E1 -20664.231,E2 -20664.231} C_VEL
LIN {X 0,Y 229.47,Z 256.493,A -85,B 0,C 180,E1 -20665.819,E2 -20665.819} C_VEL
LIN {X 0,Y 226.541,Z 252.095,A -85,B 0,C 180,E1 -20667.166,E2 -20667.166} C_VEL
LIN {X 0,Y 223.01,Z 247.506,A -85,B 0,C 180,E1 -20668.865,E2 -20668.865} C_VEL
LIN {X 0,Y 222.32,Z 246.465,A -85,B 0,C 180,E1 -20669.222,E2 -20669.222} C_VEL
LIN {X 0,Y 219.7,Z 243.938,A -85,B 0,C 180,E1 -20670.541,E2 -20670.541} C_VEL
LIN {X 0,Y 218.278,Z 241.22,A -85,B 0,C 180,E1 -20671.384,E2 -20671.384} C_VEL
LIN {X 0,Y 215.676,Z 239.431,A -85,B 0,C 180,E1 -20672.792,E2 -20672.792} C_VEL
LIN {X 0,Y 214.162,Z 236.901,A -85,B 0,C 180,E1 -20673.769,E2 -20673.769} C_VEL
LIN {X 0,Y 213.813,Z 235.47,A -85,B 0,C 180,E1 -20674.116,E2 -20674.116} C_VEL
LIN {X 0,Y 213.798,Z 235.44,A -85,B 0,C 180,E1 -20678.802,E2 -20678.802} C_VEL
LIN {X 0,Y 213.939,Z 235.454,A -85,B 0,C 180,E1 -20682.803,E2 -20682.803} C_VEL
LIN {X 0,Y 213.947,Z 235.452,A -85,B 0,C 180,E1 -20686.706,E2 -20686.706} C_VEL
LIN {X 0,Y 214.137,Z 235.43,A -85,B 0,C 180,E1 -20690.555,E2 -20690.555} C_VEL
LIN {X 0,Y 214.096,Z 235.438,A -85,B 0,C 180,E1 -20694.349,E2 -20694.349} C_VEL
LIN {X 0,Y 214.441,Z 235.399,A -85,B 0,C 180,E1 -20698.122,E2 -20698.122} C_VEL
LIN {X 0,Y 214.546,Z 235.373,A -85,B 0,C 180,E1 -20700,E2 -20700} C_VEL
LIN {X 0,Y 214.441,Z 235.398,A -85,B 0,C 180,E1 -20701.878,E2 -20701.878} C_VEL
LIN {X 0,Y 214.204,Z 235.421,A -85,B 0,C 180,E1 -20707.541,E2 -20707.541} C_VEL
LIN {X 0,Y 214.003,Z 235.45,A -85,B 0,C 180,E1 -20711.364,E2 -20711.364} C_VEL
LIN {X 0,Y 213.926,Z 235.462,A -85,B 0,C 180,E1 -20715.238,E2 -20715.238} C_VEL
LIN {X 0,Y 213.832,Z 235.474,A -85,B 0,C 180,E1 -20719.188,E2 -20719.188} C_VEL
LIN {X 0,Y 213.808,Z 235.471,A -85,B 0,C 180,E1 -20723.232,E2 -20723.232} C_VEL
LIN {X 0,Y 213.855,Z 235.494,A -85,B 0,C 180,E1 -20726.403,E2 -20726.403} C_VEL
LIN {X 0,Y 214.639,Z 237.897,A -85,B 0,C 180,E1 -20727.001,E2 -20727.001} C_VEL
LIN {X 0,Y 216.251,Z 240.001,A -85,B 0,C 180,E1 -20727.983,E2 -20727.983} C_VEL
LIN {X 0,Y 218.382,Z 241.5,A -85,B 0,C 180,E1 -20729.127,E2 -20729.127} C_VEL
LIN {X 0,Y 220.2,Z 244.623,A -85,B 0,C 180,E1 -20730.173,E2 -20730.173} C_VEL
LIN {X 0,Y 222.7,Z 246.942,A -85,B 0,C 180,E1 -20731.413,E2 -20731.413} C_VEL
LIN {X 0,Y 225.055,Z 250.365,A -85,B 0,C 180,E1 -20732.59,E2 -20732.59} C_VEL
LIN {X 0,Y 226.794,Z 252.219,A -85,B 0,C 180,E1 -20733.382,E2 -20733.382} C_VEL
LIN {X 0,Y 229.808,Z 256.105,A -85,B 0,C 180,E1 -20734.726,E2 -20734.726} C_VEL
LIN {X 0,Y 237.02,Z 266.102,A -85,B 0,C 180,E1 -20737.677,E2 -20737.677} C_VEL
LIN {X 0,Y 244.299,Z 276.912,A -85,B 0,C 180,E1 -20740.337,E2 -20740.337} C_VEL
LIN {X 0,Y 251.99,Z 289.558,A -85,B 0,C 180,E1 -20742.894,E2 -20742.894} C_VEL
LIN {X 0,Y 256.151,Z 297.791,A -85,B 0,C 180,E1 -20744.221,E2 -20744.221} C_VEL
LIN {X 0,Y 259.211,Z 304.714,A -85,B 0,C 180,E1 -20745.183,E2 -20745.183} C_VEL
LIN {X 0,Y 254.062,Z 392.224,A -85,B 0,C 180,E1 -20747.469,E2 -20747.469} C_VEL
LIN {X 0,Y 252.218,Z 408.133,A -85,B 0,C 180,E1 -20748.164,E2 -20748.164} C_VEL
LIN {X 0,Y 249.761,Z 423.242,A -85,B 0,C 180,E1 -20749.14,E2 -20749.14} C_VEL
LIN {X 0,Y 246.701,Z 437.875,A -85,B 0,C 180,E1 -20750.419,E2 -20750.419} C_VEL
LIN {X 0,Y 243.462,Z 450.984,A -85,B 0,C 180,E1 -20751.901,E2 -20751.901} C_VEL
LIN {X 0,Y 239.412,Z 464.429,A -85,B 0,C 180,E1 -20753.789,E2 -20753.789} C_VEL
LIN {X 0,Y 235.264,Z 476.63,A -85,B 0,C 180,E1 -20755.937,E2 -20755.937} C_VEL
LIN {X 0,Y 230.945,Z 487.917,A -85,B 0,C 180,E1 -20758.388,E2 -20758.388} C_VEL
LIN {X 0,Y 227.402,Z 497.084,A -85,B 0,C 180,E1 -20760.873,E2 -20760.873} C_VEL
LIN {X 0,Y 223.436,Z 506.271,A -85,B 0,C 180,E1 -20763.874,E2 -20763.874} C_VEL
LIN {X 0,Y 220.1,Z 513.902,A -85,B 0,C 180,E1 -20766.974,E2 -20766.974} C_VEL
LIN {X 0,Y 217.352,Z 520.229,A -85,B 0,C 180,E1 -20770.153,E2 -20770.153} C_VEL
LIN {X 0,Y 214.973,Z 526.034,A -85,B 0,C 180,E1 -20773.866,E2 -20773.866} C_VEL
LIN {X 0,Y 213.627,Z 529.469,A -85,B 0,C 180,E1 -20776.686,E2 -20776.686} C_VEL
LIN {X 0,Y 212.437,Z 532.943,A -85,B 0,C 180,E1 -20780.479,E2 -20780.479} C_VEL
LIN {X 0,Y 211.74,Z 535.412,A -85,B 0,C 180,E1 -20784.718,E2 -20784.718} C_VEL
LIN {X 0,Y 211.558,Z 536.399,A -85,B 0,C 180,E1 -20788.096,E2 -20788.096} C_VEL
LIN {X 0,Y 211.577,Z 536.554,A -85,B 0,C 180,E1 -20790,E2 -20790} C_VEL
LIN {X 0,Y 211.616,Z 535.993,A -85,B 0,C 180,E1 -20793.808,E2 -20793.808} C_VEL
LIN {X 0,Y 212.05,Z 534.318,A -85,B 0,C 180,E1 -20797.618,E2 -20797.618} C_VEL
LIN {X 0,Y 212.933,Z 531.49,A -85,B 0,C 180,E1 -20801.422,E2 -20801.422} C_VEL
LIN {X 0,Y 214.396,Z 527.438,A -85,B 0,C 180,E1 -20805.203,E2 -20805.203} C_VEL
LIN {X 0,Y 216.682,Z 522.056,A -85,B 0,C 180,E1 -20808.926,E2 -20808.926} C_VEL
LIN {X 0,Y 219.597,Z 515.196,A -85,B 0,C 180,E1 -20812.584,E2 -20812.584} C_VEL
LIN {X 0,Y 223.362,Z 506.625,A -85,B 0,C 180,E1 -20816.135,E2 -20816.135} C_VEL
LIN {X 0,Y 227.283,Z 497.506,A -85,B 0,C 180,E1 -20819.144,E2 -20819.144} C_VEL
LIN {X 0,Y 230.834,Z 488.384,A -85,B 0,C 180,E1 -20821.629,E2 -20821.629} C_VEL
LIN {X 0,Y 235.525,Z 476.187,A -85,B 0,C 180,E1 -20824.278,E2 -20824.278} C_VEL
LIN {X 0,Y 239.626,Z 463.898,A -85,B 0,C 180,E1 -20826.434,E2 -20826.434} C_VEL
LIN {X 0,Y 243.761,Z 450.324,A -85,B 0,C 180,E1 -20828.306,E2 -20828.306} C_VEL
LIN {X 0,Y 247.124,Z 436.588,A -85,B 0,C 180,E1 -20829.838,E2 -20829.838} C_VEL
LIN {X 0,Y 250.101,Z 422.218,A -85,B 0,C 180,E1 -20831.059,E2 -20831.059} C_VEL
LIN {X 0,Y 252.519,Z 406.681,A -85,B 0,C 180,E1 -20832.043,E2 -20832.043} C_VEL
LIN {X 0,Y 254.273,Z 391.195,A -85,B 0,C 180,E1 -20832.689,E2 -20832.689} C_VEL
LIN {X 0,Y 258.954,Z 311.186,A -85,B 0,C 180,E1 -20834.777,E2 -20834.777} C_VEL
LIN {X 0,Y 259.237,Z 304.613,A -85,B 0,C 180,E1 -20834.967,E2 -20834.967} C_VEL
LIN {X 0,Y 253.726,Z 292.518,A -85,B 0,C 180,E1 -20836.721,E2 -20836.721} C_VEL
LIN {X 0,Y 246.101,Z 279.678,A -85,B 0,C 180,E1 -20839.213,E2 -20839.213} C_VEL
LIN {X 0,Y 238.807,Z 268.553,A -85,B 0,C 180,E1 -20841.828,E2 -20841.828} C_VEL
LIN {X 0,Y 232.31,Z 259.568,A -85,B 0,C 180,E1 -20844.396,E2 -20844.396} C_VEL
LIN {X 0,Y 229.466,Z 255.675,A -85,B 0,C 180,E1 -20845.618,E2 -20845.618} C_VEL
LIN {X 0,Y 226.046,Z 251.271,A -85,B 0,C 180,E1 -20847.169,E2 -20847.169} C_VEL
LIN {X 0,Y 223.374,Z 248.108,A -85,B 0,C 180,E1 -20848.445,E2 -20848.445} C_VEL
LIN {X 0,Y 222.356,Z 246.453,A -85,B 0,C 180,E1 -20848.98,E2 -20848.98} C_VEL
LIN {X 0,Y 219.766,Z 244.007,A -85,B 0,C 180,E1 -20850.288,E2 -20850.288} C_VEL
LIN {X 0,Y 218.155,Z 241.165,A -85,B 0,C 180,E1 -20851.235,E2 -20851.235} C_VEL
LIN {X 0,Y 215.58,Z 239.338,A -85,B 0,C 180,E1 -20852.647,E2 -20852.647} C_VEL
LIN {X 0,Y 214.245,Z 237.082,A -85,B 0,C 180,E1 -20853.517,E2 -20853.517} C_VEL
LIN {X 0,Y 213.825,Z 235.465,A -85,B 0,C 180,E1 -20853.921,E2 -20853.921} C_VEL
LIN {X 0,Y 213.849,Z 235.462,A -85,B 0,C 180,E1 -20856.952,E2 -20856.952} C_VEL
LIN {X 0,Y 213.94,Z 235.455,A -85,B 0,C 180,E1 -20862.803,E2 -20862.803} C_VEL
LIN {X 0,Y 213.975,Z 235.446,A -85,B 0,C 180,E1 -20866.708,E2 -20866.708} C_VEL
LIN {X 0,Y 214.163,Z 235.419,A -85,B 0,C 180,E1 -20870.556,E2 -20870.556} C_VEL
LIN {X 0,Y 214.234,Z 235.425,A -85,B 0,C 180,E1 -20872.46,E2 -20872.46} C_VEL
LIN {X 0,Y 214.441,Z 235.391,A -85,B 0,C 180,E1 -20878.122,E2 -20878.122} C_VEL
LIN {X 0,Y 214.546,Z 235.372,A -85,B 0,C 180,E1 -20880,E2 -20880} C_VEL
LIN {X 0,Y 214.44,Z 235.399,A -85,B 0,C 180,E1 -20881.878,E2 -20881.878} C_VEL
LIN {X 0,Y 214.193,Z 235.421,A -85,B 0,C 180,E1 -20887.541,E2 -20887.541} C_VEL
LIN {X 0,Y 214.003,Z 235.453,A -85,B 0,C 180,E1 -20891.364,E2 -20891.364} C_VEL
LIN {X 0,Y 213.926,Z 235.467,A -85,B 0,C 180,E1 -20895.237,E2 -20895.237} C_VEL
LIN {X 0,Y 213.885,Z 235.461,A -85,B 0,C 180,E1 -20898.291,E2 -20898.291} C_VEL
LIN {X 0,Y 213.205,Z 235.848,A -85,B 0,C 180,E1 -20899.363,E2 -20899.363} C_VEL
LIN {X 0,Y 210.712,Z 237.595,A -85,B 0,C 180,E1 -20901.044,E2 -20901.044} C_VEL
LIN {X 0,Y 209.16,Z 239.417,A -85,B 0,C 180,E1 -20902.374,E2 -20902.374} C_VEL
LIN {X 0,Y 209.166,Z 240.744,A -85,B 0,C 180,E1 -20903.394,E2 -20903.394} C_VEL
LIN {X 0,Y 209.529,Z 241.122,A -85,B 0,C 180,E1 -20903.724,E2 -20903.724} C_VEL
LIN {X 0,Y 211.597,Z 242.36,A -85,B 0,C 180,E1 -20905.054,E2 -20905.054} C_VEL
LIN {X 0,Y 213.278,Z 245.4,A -85,B 0,C 180,E1 -20906.223,E2 -20906.223} C_VEL
LIN {X 0,Y 215.733,Z 247.582,A -85,B 0,C 180,E1 -20907.66,E2 -20907.66} C_VEL
LIN {X 0,Y 216.36,Z 248.46,A -85,B 0,C 180,E1 -20908.033,E2 -20908.033} C_VEL
LIN {X 0,Y 218.81,Z 251.812,A -85,B 0,C 180,E1 -20909.426,E2 -20909.426} C_VEL
LIN {X 0,Y 220.347,Z 253.321,A -85,B 0,C 180,E1 -20910.217,E2 -20910.217} C_VEL
LIN {X 0,Y 224.992,Z 259.736,A -85,B 0,C 180,E1 -20912.55,E2 -20912.55} C_VEL
LIN {X 0,Y 229.069,Z 266.083,A -85,B 0,C 180,E1 -20914.449,E2 -20914.449} C_VEL
LIN {X 0,Y 232.13,Z 270.985,A -85,B 0,C 180,E1 -20915.782,E2 -20915.782} C_VEL
LIN {X 0,Y 238.945,Z 282.752,A -85,B 0,C 180,E1 -20918.535,E2 -20918.535} C_VEL
LIN {X 0,Y 245.281,Z 295.023,A -85,B 0,C 180,E1 -20920.884,E2 -20920.884} C_VEL
LIN {X 0,Y 251.396,Z 308.605,A -85,B 0,C 180,E1 -20923.018,E2 -20923.018} C_VEL
LIN {X 0,Y 253.836,Z 314.577,A -85,B 0,C 180,E1 -20923.84,E2 -20923.84} C_VEL
LIN {X 0,Y 248.668,Z 400.566,A -85,B 0,C 180,E1 -20926.108,E2 -20926.108} C_VEL
LIN {X 0,Y 246.908,Z 415.554,A -85,B 0,C 180,E1 -20926.702,E2 -20926.702} C_VEL
LIN {X 0,Y 244.313,Z 430.944,A -85,B 0,C 180,E1 -20927.608,E2 -20927.608} C_VEL
LIN {X 0,Y 241.115,Z 445.192,A -85,B 0,C 180,E1 -20928.742,E2 -20928.742} C_VEL
LIN {X 0,Y 237.605,Z 458.57,A -85,B 0,C 180,E1 -20930.152,E2 -20930.152} C_VEL
LIN {X 0,Y 233.572,Z 471.763,A -85,B 0,C 180,E1 -20931.916,E2 -20931.916} C_VEL
LIN {X 0,Y 228.98,Z 484.622,A -85,B 0,C 180,E1 -20934.057,E2 -20934.057} C_VEL
LIN {X 0,Y 224.822,Z 495.395,A -85,B 0,C 180,E1 -20936.299,E2 -20936.299} C_VEL
LIN {X 0,Y 220.67,Z 505.367,A -85,B 0,C 180,E1 -20938.834,E2 -20938.834} C_VEL
LIN {X 0,Y 217.072,Z 513.875,A -85,B 0,C 180,E1 -20941.475,E2 -20941.475} C_VEL
LIN {X 0,Y 213.386,Z 522.204,A -85,B 0,C 180,E1 -20944.65,E2 -20944.65} C_VEL
LIN {X 0,Y 209.968,Z 530.034,A -85,B 0,C 180,E1 -20948.397,E2 -20948.397} C_VEL
LIN {X 0,Y 207.459,Z 536.273,A -85,B 0,C 180,E1 -20952.249,E2 -20952.249} C_VEL
LIN {X 0,Y 205.68,Z 541.104,A -85,B 0,C 180,E1 -20956.162,E2 -20956.162} C_VEL
LIN {X 0,Y 204.666,Z 544.65,A -85,B 0,C 180,E1 -20960.114,E2 -20960.114} C_VEL
LIN {X 0,Y 204.286,Z 546.988,A -85,B 0,C 180,E1 -20964.076,E2 -20964.076} C_VEL
LIN {X 0,Y 204.329,Z 548.167,A -85,B 0,C 180,E1 -20968.029,E2 -20968.029} C_VEL
LIN {X 0,Y 204.461,Z 548.325,A -85,B 0,C 180,E1 -20970,E2 -20970} C_VEL
LIN {X 0,Y 204.259,Z 547.706,A -85,B 0,C 180,E1 -20973.946,E2 -20973.946} C_VEL
LIN {X 0,Y 204.414,Z 545.932,A -85,B 0,C 180,E1 -20977.904,E2 -20977.904} C_VEL
LIN {X 0,Y 205.066,Z 542.983,A -85,B 0,C 180,E1 -20981.866,E2 -20981.866} C_VEL
LIN {X 0,Y 206.445,Z 538.793,A -85,B 0,C 180,E1 -20985.803,E2 -20985.803} C_VEL
LIN {X 0,Y 208.544,Z 533.253,A -85,B 0,C 180,E1 -20989.694,E2 -20989.694} C_VEL
LIN {X 0,Y 211.547,Z 526.218,A -85,B 0,C 180,E1 -20993.494,E2 -20993.494} C_VEL
LIN {X 0,Y 215.492,Z 517.478,A -85,B 0,C 180,E1 -20997.167,E2 -20997.167} C_VEL
LIN {X 0,Y 219.373,Z 508.311,A -85,B 0,C 180,E1 -21000.26,E2 -21000.26} C_VEL
LIN {X 0,Y 223.366,Z 498.764,A -85,B 0,C 180,E1 -21002.871,E2 -21002.871} C_VEL
LIN {X 0,Y 228.127,Z 486.534,A -85,B 0,C 180,E1 -21005.554,E2 -21005.554} C_VEL
LIN {X 0,Y 232.692,Z 474.073,A -85,B 0,C 180,E1 -21007.705,E2 -21007.705} C_VEL
LIN {X 0,Y 236.847,Z 460.802,A -85,B 0,C 180,E1 -21009.549,E2 -21009.549} C_VEL
LIN {X 0,Y 240.641,Z 446.726,A -85,B 0,C 180,E1 -21011.079,E2 -21011.079} C_VEL
LIN {X 0,Y 243.743,Z 432.929,A -85,B 0,C 180,E1 -21012.235,E2 -21012.235} C_VEL
LIN {X 0,Y 246.523,Z 417.474,A -85,B 0,C 180,E1 -21013.172,E2 -21013.172} C_VEL
LIN {X 0,Y 248.408,Z 402.166,A -85,B 0,C 180,E1 -21013.809,E2 -21013.809} C_VEL
LIN {X 0,Y 253.746,Z 314.531,A -85,B 0,C 180,E1 -21016.117,E2 -21016.117} C_VEL
LIN {X 0,Y 248.676,Z 302.476,A -85,B 0,C 180,E1 -21017.839,E2 -21017.839} C_VEL
LIN {X 0,Y 242.389,Z 289.328,A -85,B 0,C 180,E1 -21020.083,E2 -21020.083} C_VEL
LIN {X 0,Y 235.679,Z 277.103,A -85,B 0,C 180,E1 -21022.652,E2 -21022.652} C_VEL
LIN {X 0,Y 230.321,Z 267.969,A -85,B 0,C 180,E1 -21024.901,E2 -21024.901} C_VEL
LIN {X 0,Y 226.342,Z 261.872,A -85,B 0,C 180,E1 -21026.69,E2 -21026.69} C_VEL
LIN {X 0,Y 223.615,Z 257.713,A -85,B 0,C 180,E1 -21028.004,E2 -21028.004} C_VEL
LIN {X 0,Y 220.351,Z 253.354,A -85,B 0,C 180,E1 -21029.649,E2 -21029.649} C_VEL
LIN {X 0,Y 216.96,Z 249.518,A -85,B 0,C 180,E1 -21031.459,E2 -21031.459} C_VEL
LIN {X 0,Y 215.807,Z 247.613,A -85,B 0,C 180,E1 -21032.153,E2 -21032.153} C_VEL
LIN {X 0,Y 213.23,Z 245.339,A -85,B 0,C 180,E1 -21033.648,E2 -21033.648} C_VEL
LIN {X 0,Y 211.376,Z 242.153,A -85,B 0,C 180,E1 -21034.918,E2 -21034.918} C_VEL
LIN {X 0,Y 208.778,Z 240.472,A -85,B 0,C 180,E1 -21036.612,E2 -21036.612} C_VEL
LIN {X 0,Y 207.182,Z 238.015,A -85,B 0,C 180,E1 -21037.861,E2 -21037.861} C_VEL
LIN {X 0,Y 206.756,Z 236.315,A -85,B 0,C 180,E1 -21038.371,E2 -21038.371} C_VEL
LIN {X 0,Y 206.869,Z 236.34,A -85,B 0,C 180,E1 -21042.196,E2 -21042.196} C_VEL
LIN {X 0,Y 206.89,Z 236.335,A -85,B 0,C 180,E1 -21046.244,E2 -21046.244} C_VEL
LIN {X 0,Y 207.096,Z 236.309,A -85,B 0,C 180,E1 -21050.231,E2 -21050.231} C_VEL
LIN {X 0,Y 207.057,Z 236.317,A -85,B 0,C 180,E1 -21054.156,E2 -21054.156} C_VEL
LIN {X 0,Y 207.377,Z 236.279,A -85,B 0,C 180,E1 -21058.058,E2 -21058.058} C_VEL
LIN {X 0,Y 207.511,Z 236.249,A -85,B 0,C 180,E1 -21060,E2 -21060} C_VEL
LIN {X 0,Y 207.377,Z 236.278,A -85,B 0,C 180,E1 -21061.942,E2 -21061.942} C_VEL
LIN {X 0,Y 207.144,Z 236.298,A -85,B 0,C 180,E1 -21067.8,E2 -21067.8} C_VEL
LIN {X 0,Y 206.926,Z 236.327,A -85,B 0,C 180,E1 -21071.758,E2 -21071.758} C_VEL
LIN {X 0,Y 206.86,Z 236.337,A -85,B 0,C 180,E1 -21075.771,E2 -21075.771} C_VEL
LIN {X 0,Y 206.759,Z 236.348,A -85,B 0,C 180,E1 -21079.872,E2 -21079.872} C_VEL
LIN {X 0,Y 206.752,Z 236.457,A -85,B 0,C 180,E1 -21082.15,E2 -21082.15} C_VEL
LIN {X 0,Y 207.516,Z 238.74,A -85,B 0,C 180,E1 -21082.87,E2 -21082.87} C_VEL
LIN {X 0,Y 209.249,Z 240.934,A -85,B 0,C 180,E1 -21084.164,E2 -21084.164} C_VEL
LIN {X 0,Y 211.574,Z 242.244,A -85,B 0,C 180,E1 -21085.646,E2 -21085.646} C_VEL
LIN {X 0,Y 213.294,Z 245.441,A -85,B 0,C 180,E1 -21086.837,E2 -21086.837} C_VEL
LIN {X 0,Y 215.836,Z 247.633,A -85,B 0,C 180,E1 -21088.306,E2 -21088.306} C_VEL
LIN {X 0,Y 218.435,Z 251.452,A -85,B 0,C 180,E1 -21089.808,E2 -21089.808} C_VEL
LIN {X 0,Y 220.379,Z 253.47,A -85,B 0,C 180,E1 -21090.813,E2 -21090.813} C_VEL
LIN {X 0,Y 223.176,Z 257.151,A -85,B 0,C 180,E1 -21092.227,E2 -21092.227} C_VEL
LIN {X 0,Y 224.741,Z 259.201,A -85,B 0,C 180,E1 -21092.978,E2 -21092.978} C_VEL
LIN {X 0,Y 228.084,Z 263.632,A -85,B 0,C 180,E1 -21094.505,E2 -21094.505} C_VEL
LIN {X 0,Y 233.763,Z 271.521,A -85,B 0,C 180,E1 -21096.895,E2 -21096.895} C_VEL
LIN {X 0,Y 240.961,Z 282.506,A -85,B 0,C 180,E1 -21099.644,E2 -21099.644} C_VEL
LIN {X 0,Y 248.131,Z 294.464,A -85,B 0,C 180,E1 -21102.127,E2 -21102.127} C_VEL
LIN {X 0,Y 252.296,Z 302.982,A -85,B 0,C 180,E1 -21103.518,E2 -21103.518} C_VEL
LIN {X 0,Y 254.06,Z 306.983,A -85,B 0,C 180,E1 -21104.099,E2 -21104.099} C_VEL
LIN {X 0,Y 248.99,Z 391.072,A -85,B 0,C 180,E1 -21106.319,E2 -21106.319} C_VEL
LIN {X 0,Y 247.221,Z 406.696,A -85,B 0,C 180,E1 -21106.98,E2 -21106.98} C_VEL
LIN {X 0,Y 244.654,Z 422.291,A -85,B 0,C 180,E1 -21107.959,E2 -21107.959} C_VEL
LIN {X 0,Y 241.634,Z 436.535,A -85,B 0,C 180,E1 -21109.186,E2 -21109.186} C_VEL
LIN {X 0,Y 237.91,Z 451.189,A -85,B 0,C 180,E1 -21110.845,E2 -21110.845} C_VEL
LIN {X 0,Y 233.709,Z 464.634,A -85,B 0,C 180,E1 -21112.758,E2 -21112.758} C_VEL
LIN {X 0,Y 229.408,Z 476.834,A -85,B 0,C 180,E1 -21114.942,E2 -21114.942} C_VEL
LIN {X 0,Y 224.918,Z 488.121,A -85,B 0,C 180,E1 -21117.438,E2 -21117.438} C_VEL
LIN {X 0,Y 220.557,Z 498.734,A -85,B 0,C 180,E1 -21120.403,E2 -21120.403} C_VEL
LIN {X 0,Y 216.53,Z 507.689,A -85,B 0,C 180,E1 -21123.495,E2 -21123.495} C_VEL
LIN {X 0,Y 213.078,Z 515.105,A -85,B 0,C 180,E1 -21126.685,E2 -21126.685} C_VEL
LIN {X 0,Y 209.954,Z 522.03,A -85,B 0,C 180,E1 -21130.444,E2 -21130.444} C_VEL
LIN {X 0,Y 207.546,Z 527.466,A -85,B 0,C 180,E1 -21134.283,E2 -21134.283} C_VEL
LIN {X 0,Y 205.971,Z 531.561,A -85,B 0,C 180,E1 -21138.187,E2 -21138.187} C_VEL
LIN {X 0,Y 205.011,Z 534.433,A -85,B 0,C 180,E1 -21142.119,E2 -21142.119} C_VEL
LIN {X 0,Y 204.54,Z 536.157,A -85,B 0,C 180,E1 -21146.06,E2 -21146.06} C_VEL
LIN {X 0,Y 204.496,Z 536.754,A -85,B 0,C 180,E1 -21150,E2 -21150} C_VEL
LIN {X 0,Y 204.553,Z 536.193,A -85,B 0,C 180,E1 -21153.94,E2 -21153.94} C_VEL
LIN {X 0,Y 205.002,Z 534.518,A -85,B 0,C 180,E1 -21157.882,E2 -21157.882} C_VEL
LIN {X 0,Y 205.939,Z 531.691,A -85,B 0,C 180,E1 -21161.815,E2 -21161.815} C_VEL
LIN {X 0,Y 207.52,Z 527.638,A -85,B 0,C 180,E1 -21165.719,E2 -21165.719} C_VEL
LIN {X 0,Y 209.931,Z 522.257,A -85,B 0,C 180,E1 -21169.558,E2 -21169.558} C_VEL
LIN {X 0,Y 213.014,Z 515.397,A -85,B 0,C 180,E1 -21173.323,E2 -21173.323} C_VEL
LIN {X 0,Y 217,Z 506.824,A -85,B 0,C 180,E1 -21176.963,E2 -21176.963} C_VEL
LIN {X 0,Y 221.092,Z 497.705,A -85,B 0,C 180,E1 -21180.043,E2 -21180.043} C_VEL
LIN {X 0,Y 224.879,Z 488.419,A -85,B 0,C 180,E1 -21182.622,E2 -21182.622} C_VEL
LIN {X 0,Y 229.691,Z 476.384,A -85,B 0,C 180,E1 -21185.276,E2 -21185.276} C_VEL
LIN {X 0,Y 233.534,Z 465.28,A -85,B 0,C 180,E1 -21187.274,E2 -21187.274} C_VEL
LIN {X 0,Y 237.798,Z 451.987,A -85,B 0,C 180,E1 -21189.177,E2 -21189.177} C_VEL
LIN {X 0,Y 241.115,Z 439.28,A -85,B 0,C 180,E1 -21190.653,E2 -21190.653} C_VEL
LIN {X 0,Y 244.307,Z 424.689,A -85,B 0,C 180,E1 -21191.976,E2 -21191.976} C_VEL
LIN {X 0,Y 246.828,Z 410.009,A -85,B 0,C 180,E1 -21192.966,E2 -21192.966} C_VEL
LIN {X 0,Y 248.769,Z 394.95,A -85,B 0,C 180,E1 -21193.659,E2 -21193.659} C_VEL
LIN {X 0,Y 250.335,Z 373.017,A -85,B 0,C 180,E1 -21194.293,E2 -21194.293} C_VEL
LIN {X 0,Y 254.016,Z 310.297,A -85,B 0,C 180,E1 -21195.936,E2 -21195.936} C_VEL
LIN {X 0,Y 254.097,Z 306.935,A -85,B 0,C 180,E1 -21196.051,E2 -21196.051} C_VEL
LIN {X 0,Y 248.892,Z 295.705,A -85,B 0,C 180,E1 -21197.788,E2 -21197.788} C_VEL
LIN {X 0,Y 242.118,Z 284.246,A -85,B 0,C 180,E1 -21200.117,E2 -21200.117} C_VEL
LIN {X 0,Y 235.042,Z 273.371,A -85,B 0,C 180,E1 -21202.779,E2 -21202.779} C_VEL
LIN {X 0,Y 229.142,Z 265.016,A -85,B 0,C 180,E1 -21205.229,E2 -21205.229} C_VEL
LIN {X 0,Y 226.402,Z 261.272,A -85,B 0,C 180,E1 -21206.459,E2 -21206.459} C_VEL
LIN {X 0,Y 223.315,Z 257.236,A -85,B 0,C 180,E1 -21207.921,E2 -21207.921} C_VEL
LIN {X 0,Y 220.51,Z 253.602,A -85,B 0,C 180,E1 -21209.34,E2 -21209.34} C_VEL
LIN {X 0,Y 219.451,Z 252.338,A -85,B 0,C 180,E1 -21209.894,E2 -21209.894} C_VEL
LIN {X 0,Y 216.948,Z 249.447,A -85,B 0,C 180,E1 -21211.258,E2 -21211.258} C_VEL
LIN {X 0,Y 215.995,Z 247.677,A -85,B 0,C 180,E1 -21211.849,E2 -21211.849} C_VEL
LIN {X 0,Y 213.462,Z 245.621,A -85,B 0,C 180,E1 -21213.308,E2 -21213.308} C_VEL
LIN {X 0,Y 211.798,Z 242.782,A -85,B 0,C 180,E1 -21214.445,E2 -21214.445} C_VEL
LIN {X 0,Y 211.491,Z 242.164,A -85,B 0,C 180,E1 -21214.669,E2 -21214.669} C_VEL
LIN {X 0,Y 208.884,Z 240.575,A -85,B 0,C 180,E1 -21216.372,E2 -21216.372} C_VEL
LIN {X 0,Y 207.197,Z 238.017,A -85,B 0,C 180,E1 -21217.701,E2 -21217.701} C_VEL
LIN {X 0,Y 206.752,Z 236.347,A -85,B 0,C 180,E1 -21218.174,E2 -21218.174} C_VEL
LIN {X 0,Y 206.87,Z 236.331,A -85,B 0,C 180,E1 -21222.196,E2 -21222.196} C_VEL
LIN {X 0,Y 206.908,Z 236.324,A -85,B 0,C 180,E1 -21226.245,E2 -21226.245} C_VEL
LIN {X 0,Y 207.101,Z 236.298,A -85,B 0,C 180,E1 -21230.231,E2 -21230.231} C_VEL
LIN {X 0,Y 207.173,Z 236.304,A -85,B 0,C 180,E1 -21232.201,E2 -21232.201} C_VEL
LIN {X 0,Y 207.377,Z 236.271,A -85,B 0,C 180,E1 -21238.058,E2 -21238.058} C_VEL
LIN {X 0,Y 207.51,Z 236.248,A -85,B 0,C 180,E1 -21240,E2 -21240} C_VEL
LIN {X 0,Y 207.377,Z 236.28,A -85,B 0,C 180,E1 -21241.942,E2 -21241.942} C_VEL
LIN {X 0,Y 207.136,Z 236.298,A -85,B 0,C 180,E1 -21247.8,E2 -21247.8} C_VEL
LIN {X 0,Y 206.925,Z 236.33,A -85,B 0,C 180,E1 -21251.758,E2 -21251.758} C_VEL
LIN {X 0,Y 206.86,Z 236.343,A -85,B 0,C 180,E1 -21255.771,E2 -21255.771} C_VEL
LIN {X 0,Y 206.795,Z 236.353,A -85,B 0,C 180,E1 -21259.868,E2 -21259.868} C_VEL
LIN {X 0,Y 206.762,Z 236.378,A -85,B 0,C 180,E1 -21261.497,E2 -21261.497} C_VEL
LIN {X 0,Y 207.47,Z 238.676,A -85,B 0,C 180,E1 -21262.19,E2 -21262.19} C_VEL
LIN {X 0,Y 209.529,Z 241.122,A -85,B 0,C 180,E1 -21263.724,E2 -21263.724} C_VEL
LIN {X 0,Y 210.78,Z 242.84,A -85,B 0,C 180,E1 -21264.617,E2 -21264.617} C_VEL
LIN {X 0,Y 212.02,Z 246.459,A -85,B 0,C 180,E1 -21265.61,E2 -21265.61} C_VEL
LIN {X 0,Y 213.928,Z 253.844,A -85,B 0,C 180,E1 -21267.182,E2 -21267.182} C_VEL
LIN {X 0,Y 214.673,Z 255.669,A -85,B 0,C 180,E1 -21267.692,E2 -21267.692} C_VEL
LIN {X 0,Y 217.453,Z 258.944,A -85,B 0,C 180,E1 -21269.263,E2 -21269.263} C_VEL
LIN {X 0,Y 222.248,Z 265.571,A -85,B 0,C 180,E1 -21271.783,E2 -21271.783} C_VEL
LIN {X 0,Y 228.171,Z 274.961,A -85,B 0,C 180,E1 -21274.604,E2 -21274.604} C_VEL
LIN {X 0,Y 235.356,Z 287.778,A -85,B 0,C 180,E1 -21277.677,E2 -21277.677} C_VEL
LIN {X 0,Y 241.289,Z 299.487,A -85,B 0,C 180,E1 -21279.987,E2 -21279.987} C_VEL
LIN {X 0,Y 247.081,Z 312.611,A -85,B 0,C 180,E1 -21282.111,E2 -21282.111} C_VEL
LIN {X 0,Y 248.732,Z 316.686,A -85,B 0,C 180,E1 -21282.697,E2 -21282.697} C_VEL
LIN {X 0,Y 247.601,Z 337.903,A -85,B 0,C 180,E1 -21283.298,E2 -21283.298} C_VEL
LIN {X 0,Y 243.456,Z 401.861,A -85,B 0,C 180,E1 -21284.989,E2 -21284.989} C_VEL
LIN {X 0,Y 241.429,Z 418.001,A -85,B 0,C 180,E1 -21285.683,E2 -21285.683} C_VEL
LIN {X 0,Y 238.592,Z 433.246,A -85,B 0,C 180,E1 -21286.632,E2 -21286.632} C_VEL
LIN {X 0,Y 235.336,Z 446.981,A -85,B 0,C 180,E1 -21287.785,E2 -21287.785} C_VEL
LIN {X 0,Y 231.61,Z 460.379,A -85,B 0,C 180,E1 -21289.267,E2 -21289.267} C_VEL
LIN {X 0,Y 227.113,Z 474.152,A -85,B 0,C 180,E1 -21291.199,E2 -21291.199} C_VEL
LIN {X 0,Y 222.387,Z 486.568,A -85,B 0,C 180,E1 -21293.382,E2 -21293.382} C_VEL
LIN {X 0,Y 217.429,Z 498.749,A -85,B 0,C 180,E1 -21296.113,E2 -21296.113} C_VEL
LIN {X 0,Y 212.691,Z 509.399,A -85,B 0,C 180,E1 -21299.116,E2 -21299.116} C_VEL
LIN {X 0,Y 208.598,Z 518.631,A -85,B 0,C 180,E1 -21302.403,E2 -21302.403} C_VEL
LIN {X 0,Y 205.013,Z 526.132,A -85,B 0,C 180,E1 -21305.71,E2 -21305.71} C_VEL
LIN {X 0,Y 201.845,Z 533.137,A -85,B 0,C 180,E1 -21309.624,E2 -21309.624} C_VEL
LIN {X 0,Y 199.578,Z 538.653,A -85,B 0,C 180,E1 -21313.638,E2 -21313.638} C_VEL
LIN {X 0,Y 198.059,Z 542.829,A -85,B 0,C 180,E1 -21317.708,E2 -21317.708} C_VEL
LIN {X 0,Y 197.339,Z 545.765,A -85,B 0,C 180,E1 -21321.81,E2 -21321.81} C_VEL
LIN {X 0,Y 197.171,Z 547.52,A -85,B 0,C 180,E1 -21325.912,E2 -21325.912} C_VEL
LIN {X 0,Y 197.361,Z 548.124,A -85,B 0,C 180,E1 -21330,E2 -21330} C_VEL
LIN {X 0,Y 197.171,Z 547.504,A -85,B 0,C 180,E1 -21334.088,E2 -21334.088} C_VEL
LIN {X 0,Y 197.339,Z 545.73,A -85,B 0,C 180,E1 -21338.19,E2 -21338.19} C_VEL
LIN {X 0,Y 198.057,Z 542.779,A -85,B 0,C 180,E1 -21342.293,E2 -21342.293} C_VEL
LIN {X 0,Y 199.539,Z 538.589,A -85,B 0,C 180,E1 -21346.365,E2 -21346.365} C_VEL
LIN {X 0,Y 201.808,Z 533.049,A -85,B 0,C 180,E1 -21350.38,E2 -21350.38} C_VEL
LIN {X 0,Y 205.006,Z 526.014,A -85,B 0,C 180,E1 -21354.291,E2 -21354.291} C_VEL
LIN {X 0,Y 208.591,Z 518.5,A -85,B 0,C 180,E1 -21357.598,E2 -21357.598} C_VEL
LIN {X 0,Y 212.672,Z 509.279,A -85,B 0,C 180,E1 -21360.875,E2 -21360.875} C_VEL
LIN {X 0,Y 217.404,Z 498.559,A -85,B 0,C 180,E1 -21363.892,E2 -21363.892} C_VEL
LIN {X 0,Y 222.36,Z 486.329,A -85,B 0,C 180,E1 -21366.624,E2 -21366.624} C_VEL
LIN {X 0,Y 227.107,Z 473.868,A -85,B 0,C 180,E1 -21368.802,E2 -21368.802} C_VEL
LIN {X 0,Y 231.168,Z 461.339,A -85,B 0,C 180,E1 -21370.582,E2 -21370.582} C_VEL
LIN {X 0,Y 235.338,Z 446.519,A -85,B 0,C 180,E1 -21372.215,E2 -21372.215} C_VEL
LIN {X 0,Y 238.544,Z 432.721,A -85,B 0,C 180,E1 -21373.379,E2 -21373.379} C_VEL
LIN {X 0,Y 241.386,Z 417.263,A -85,B 0,C 180,E1 -21374.327,E2 -21374.327} C_VEL
LIN {X 0,Y 243.342,Z 401.95,A -85,B 0,C 180,E1 -21374.965,E2 -21374.965} C_VEL
LIN {X 0,Y 248.728,Z 316.846,A -85,B 0,C 180,E1 -21377.227,E2 -21377.227} C_VEL
LIN {X 0,Y 243.116,Z 303.612,A -85,B 0,C 180,E1 -21379.245,E2 -21379.245} C_VEL
LIN {X 0,Y 237.154,Z 291.29,A -85,B 0,C 180,E1 -21381.514,E2 -21381.514} C_VEL
LIN {X 0,Y 230.058,Z 278.292,A -85,B 0,C 180,E1 -21384.45,E2 -21384.45} C_VEL
LIN {X 0,Y 226.138,Z 271.763,A -85,B 0,C 180,E1 -21386.213,E2 -21386.213} C_VEL
LIN {X 0,Y 221.055,Z 263.77,A -85,B 0,C 180,E1 -21388.702,E2 -21388.702} C_VEL
LIN {X 0,Y 217.787,Z 259.304,A -85,B 0,C 180,E1 -21390.422,E2 -21390.422} C_VEL
LIN {X 0,Y 214.598,Z 255.6,A -85,B 0,C 180,E1 -21392.202,E2 -21392.202} C_VEL
LIN {X 0,Y 213.503,Z 253.976,A -85,B 0,C 180,E1 -21392.875,E2 -21392.875} C_VEL
LIN {X 0,Y 210.839,Z 251.247,A -85,B 0,C 180,E1 -21394.519,E2 -21394.519} C_VEL
LIN {X 0,Y 209.514,Z 248.854,A -85,B 0,C 180,E1 -21395.474,E2 -21395.474} C_VEL
LIN {X 0,Y 206.87,Z 246.865,A -85,B 0,C 180,E1 -21397.287,E2 -21397.287} C_VEL
LIN {X 0,Y 205.068,Z 243.97,A -85,B 0,C 180,E1 -21398.778,E2 -21398.778} C_VEL
LIN {X 0,Y 204.688,Z 243.114,A -85,B 0,C 180,E1 -21399.132,E2 -21399.132} C_VEL
LIN {X 0,Y 201.961,Z 241.536,A -85,B 0,C 180,E1 -21401.408,E2 -21401.408} C_VEL
LIN {X 0,Y 200.284,Z 239.005,A -85,B 0,C 180,E1 -21403.173,E2 -21403.173} C_VEL
LIN {X 0,Y 199.824,Z 237.209,A -85,B 0,C 180,E1 -21403.921,E2 -21403.921} C_VEL
LIN {X 0,Y 200.019,Z 237.194,A -85,B 0,C 180,E1 -21409.882,E2 -21409.882} C_VEL
LIN {X 0,Y 200.018,Z 237.195,A -85,B 0,C 180,E1 -21413.949,E2 -21413.949} C_VEL
LIN {X 0,Y 200.316,Z 237.159,A -85,B 0,C 180,E1 -21417.99,E2 -21417.99} C_VEL
LIN {X 0,Y 200.475,Z 237.125,A -85,B 0,C 180,E1 -21420,E2 -21420} C_VEL
LIN {X 0,Y 200.023,Z 237.182,A -85,B 0,C 180,E1 -21424.03,E2 -21424.03} C_VEL
LIN {X 0,Y 200.091,Z 237.175,A -85,B 0,C 180,E1 -21428.077,E2 -21428.077} C_VEL
LIN {X 0,Y 199.874,Z 237.203,A -85,B 0,C 180,E1 -21432.18,E2 -21432.18} C_VEL
LIN {X 0,Y 199.809,Z 237.275,A -85,B 0,C 180,E1 -21436.606,E2 -21436.606} C_VEL
LIN {X 0,Y 200.344,Z 239.189,A -85,B 0,C 180,E1 -21437.348,E2 -21437.348} C_VEL
LIN {X 0,Y 202.092,Z 241.687,A -85,B 0,C 180,E1 -21439.16,E2 -21439.16} C_VEL
LIN {X 0,Y 204.843,Z 243.339,A -85,B 0,C 180,E1 -21441.445,E2 -21441.445} C_VEL
LIN {X 0,Y 206.365,Z 246.296,A -85,B 0,C 180,E1 -21442.772,E2 -21442.772} C_VEL
LIN {X 0,Y 208.939,Z 248.541,A -85,B 0,C 180,E1 -21444.599,E2 -21444.599} C_VEL
LIN {X 0,Y 209.644,Z 249.108,A -85,B 0,C 180,E1 -21445.066,E2 -21445.066} C_VEL
LIN {X 0,Y 211.71,Z 252.374,A -85,B 0,C 180,E1 -21446.494,E2 -21446.494} C_VEL
LIN {X 0,Y 213.958,Z 254.549,A -85,B 0,C 180,E1 -21447.843,E2 -21447.843} C_VEL
LIN {X 0,Y 216.597,Z 258.176,A -85,B 0,C 180,E1 -21449.391,E2 -21449.391} C_VEL
LIN {X 0,Y 218.143,Z 259.948,A -85,B 0,C 180,E1 -21450.225,E2 -21450.225} C_VEL
LIN {X 0,Y 222.23,Z 265.37,A -85,B 0,C 180,E1 -21452.327,E2 -21452.327} C_VEL
LIN {X 0,Y 225.673,Z 270.093,A -85,B 0,C 180,E1 -21453.96,E2 -21453.96} C_VEL
LIN {X 0,Y 230.725,Z 277.26,A -85,B 0,C 180,E1 -21456.169,E2 -21456.169} C_VEL
LIN {X 0,Y 237.491,Z 287.777,A -85,B 0,C 180,E1 -21458.865,E2 -21458.865} C_VEL
LIN {X 0,Y 244.346,Z 299.501,A -85,B 0,C 180,E1 -21461.349,E2 -21461.349} C_VEL
LIN {X 0,Y 248.18,Z 307.531,A -85,B 0,C 180,E1 -21462.691,E2 -21462.691} C_VEL
LIN {X 0,Y 249.012,Z 309.479,A -85,B 0,C 180,E1 -21462.981,E2 -21462.981} C_VEL
LIN {X 0,Y 243.921,Z 391.292,A -85,B 0,C 180,E1 -21465.171,E2 -21465.171} C_VEL
LIN {X 0,Y 242.097,Z 406.908,A -85,B 0,C 180,E1 -21465.838,E2 -21465.838} C_VEL
LIN {X 0,Y 239.439,Z 422.5,A -85,B 0,C 180,E1 -21466.823,E2 -21466.823} C_VEL
LIN {X 0,Y 236.292,Z 436.841,A -85,B 0,C 180,E1 -21468.072,E2 -21468.072} C_VEL
LIN {X 0,Y 232.458,Z 451.395,A -85,B 0,C 180,E1 -21469.742,E2 -21469.742} C_VEL
LIN {X 0,Y 228.076,Z 464.839,A -85,B 0,C 180,E1 -21471.675,E2 -21471.675} C_VEL
LIN {X 0,Y 223.607,Z 477.039,A -85,B 0,C 180,E1 -21473.893,E2 -21473.893} C_VEL
LIN {X 0,Y 219.025,Z 488.155,A -85,B 0,C 180,E1 -21476.393,E2 -21476.393} C_VEL
LIN {X 0,Y 214.404,Z 498.938,A -85,B 0,C 180,E1 -21479.465,E2 -21479.465} C_VEL
LIN {X 0,Y 210.168,Z 507.893,A -85,B 0,C 180,E1 -21482.627,E2 -21482.627} C_VEL
LIN {X 0,Y 206.552,Z 515.309,A -85,B 0,C 180,E1 -21485.902,E2 -21485.902} C_VEL
LIN {X 0,Y 203.229,Z 522.234,A -85,B 0,C 180,E1 -21489.769,E2 -21489.769} C_VEL
LIN {X 0,Y 200.693,Z 527.669,A -85,B 0,C 180,E1 -21493.731,E2 -21493.731} C_VEL
LIN {X 0,Y 198.996,Z 531.764,A -85,B 0,C 180,E1 -21497.766,E2 -21497.766} C_VEL
LIN {X 0,Y 197.959,Z 534.635,A -85,B 0,C 180,E1 -21501.836,E2 -21501.836} C_VEL
LIN {X 0,Y 197.463,Z 536.357,A -85,B 0,C 180,E1 -21505.918,E2 -21505.918} C_VEL
LIN {X 0,Y 197.397,Z 536.955,A -85,B 0,C 180,E1 -21510,E2 -21510} C_VEL
LIN {X 0,Y 197.463,Z 536.394,A -85,B 0,C 180,E1 -21514.082,E2 -21514.082} C_VEL
LIN {X 0,Y 197.95,Z 534.719,A -85,B 0,C 180,E1 -21518.164,E2 -21518.164} C_VEL
LIN {X 0,Y 198.967,Z 531.892,A -85,B 0,C 180,E1 -21522.235,E2 -21522.235} C_VEL
LIN {X 0,Y 200.668,Z 527.839,A -85,B 0,C 180,E1 -21526.271,E2 -21526.271} C_VEL
LIN {X 0,Y 203.218,Z 522.457,A -85,B 0,C 180,E1 -21530.232,E2 -21530.232} C_VEL
LIN {X 0,Y 206.487,Z 515.597,A -85,B 0,C 180,E1 -21534.106,E2 -21534.106} C_VEL
LIN {X 0,Y 210.662,Z 507.024,A -85,B 0,C 180,E1 -21537.843,E2 -21537.843} C_VEL
LIN {X 0,Y 214.3,Z 499.313,A -85,B 0,C 180,E1 -21540.551,E2 -21540.551} C_VEL
LIN {X 0,Y 218.916,Z 488.618,A -85,B 0,C 180,E1 -21543.626,E2 -21543.626} C_VEL
LIN {X 0,Y 223.929,Z 476.582,A -85,B 0,C 180,E1 -21546.326,E2 -21546.326} C_VEL
LIN {X 0,Y 227.936,Z 465.476,A -85,B 0,C 180,E1 -21548.353,E2 -21548.353} C_VEL
LIN {X 0,Y 231.899,Z 453.603,A -85,B 0,C 180,E1 -21550.09,E2 -21550.09} C_VEL
LIN {X 0,Y 235.662,Z 439.877,A -85,B 0,C 180,E1 -21551.737,E2 -21551.737} C_VEL
LIN {X 0,Y 238.848,Z 426.01,A -85,B 0,C 180,E1 -21553.021,E2 -21553.021} C_VEL
LIN {X 0,Y 241.58,Z 410.96,A -85,B 0,C 180,E1 -21554.064,E2 -21554.064} C_VEL
LIN {X 0,Y 243.579,Z 396.273,A -85,B 0,C 180,E1 -21554.763,E2 -21554.763} C_VEL
LIN {X 0,Y 245.114,Z 376.767,A -85,B 0,C 180,E1 -21555.35,E2 -21555.35} C_VEL
LIN {X 0,Y 249.127,Z 310.678,A -85,B 0,C 180,E1 -21557.102,E2 -21557.102} C_VEL
LIN {X 0,Y 248.983,Z 309.18,A -85,B 0,C 180,E1 -21557.2,E2 -21557.2} C_VEL
LIN {X 0,Y 244.784,Z 300.121,A -85,B 0,C 180,E1 -21558.673,E2 -21558.673} C_VEL
LIN {X 0,Y 237.984,Z 288.477,A -85,B 0,C 180,E1 -21561.131,E2 -21561.131} C_VEL
LIN {X 0,Y 231.385,Z 278.183,A -85,B 0,C 180,E1 -21563.747,E2 -21563.747} C_VEL
LIN {X 0,Y 224.289,Z 267.911,A -85,B 0,C 180,E1 -21566.902,E2 -21566.902} C_VEL
LIN {X 0,Y 220.628,Z 263.168,A -85,B 0,C 180,E1 -21568.693,E2 -21568.693} C_VEL
LIN {X 0,Y 217.171,Z 258.66,A -85,B 0,C 180,E1 -21570.535,E2 -21570.535} C_VEL
LIN {X 0,Y 214.451,Z 255.302,A -85,B 0,C 180,E1 -21572.093,E2 -21572.093} C_VEL
LIN {X 0,Y 213.468,Z 253.917,A -85,B 0,C 180,E1 -21572.7,E2 -21572.7} C_VEL
LIN {X 0,Y 210.859,Z 251.262,A -85,B 0,C 180,E1 -21574.323,E2 -21574.323} C_VEL
LIN {X 0,Y 209.463,Z 248.792,A -85,B 0,C 180,E1 -21575.335,E2 -21575.335} C_VEL
LIN {X 0,Y 206.803,Z 246.776,A -85,B 0,C 180,E1 -21577.184,E2 -21577.184} C_VEL
LIN {X 0,Y 205.073,Z 243.878,A -85,B 0,C 180,E1 -21578.646,E2 -21578.646} C_VEL
LIN {X 0,Y 204.831,Z 243.232,A -85,B 0,C 180,E1 -21578.883,E2 -21578.883} C_VEL
LIN {X 0,Y 201.87,Z 241.442,A -85,B 0,C 180,E1 -21581.399,E2 -21581.399} C_VEL
LIN {X 0,Y 200.184,Z 238.802,A -85,B 0,C 180,E1 -21583.229,E2 -21583.229} C_VEL
LIN {X 0,Y 199.814,Z 237.22,A -85,B 0,C 180,E1 -21583.854,E2 -21583.854} C_VEL
LIN {X 0,Y 200.067,Z 237.175,A -85,B 0,C 180,E1 -21589.884,E2 -21589.884} C_VEL
LIN {X 0,Y 200.032,Z 237.181,A -85,B 0,C 180,E1 -21593.949,E2 -21593.949} C_VEL
LIN {X 0,Y 200.317,Z 237.15,A -85,B 0,C 180,E1 -21597.989,E2 -21597.989} C_VEL
LIN {X 0,Y 200.475,Z 237.124,A -85,B 0,C 180,E1 -21600,E2 -21600} C_VEL
LIN {X 0,Y 200.022,Z 237.18,A -85,B 0,C 180,E1 -21604.029,E2 -21604.029} C_VEL
LIN {X 0,Y 200.084,Z 237.174,A -85,B 0,C 180,E1 -21608.077,E2 -21608.077} C_VEL
LIN {X 0,Y 199.873,Z 237.204,A -85,B 0,C 180,E1 -21612.179,E2 -21612.179} C_VEL
LIN {X 0,Y 199.824,Z 237.337,A -85,B 0,C 180,E1 -21615.883,E2 -21615.883} C_VEL
LIN {X 0,Y 200.452,Z 239.42,A -85,B 0,C 180,E1 -21616.747,E2 -21616.747} C_VEL
LIN {X 0,Y 202.523,Z 241.997,A -85,B 0,C 180,E1 -21618.854,E2 -21618.854} C_VEL
LIN {X 0,Y 204.848,Z 243.333,A -85,B 0,C 180,E1 -21620.786,E2 -21620.786} C_VEL
LIN {X 0,Y 206.318,Z 246.182,A -85,B 0,C 180,E1 -21622.084,E2 -21622.084} C_VEL
LIN {X 0,Y 208.975,Z 248.576,A -85,B 0,C 180,E1 -21623.999,E2 -21623.999} C_VEL
LIN {X 0,Y 209.715,Z 249.266,A -85,B 0,C 180,E1 -21624.501,E2 -21624.501} C_VEL
LIN {X 0,Y 211.843,Z 252.429,A -85,B 0,C 180,E1 -21625.965,E2 -21625.965} C_VEL
LIN {X 0,Y 214.044,Z 254.631,A -85,B 0,C 180,E1 -21627.298,E2 -21627.298} C_VEL
LIN {X 0,Y 214.673,Z 255.669,A -85,B 0,C 180,E1 -21627.692,E2 -21627.692} C_VEL
LIN {X 0,Y 216.925,Z 260.931,A -85,B 0,C 180,E1 -21629.147,E2 -21629.147} C_VEL
LIN {X 0,Y 221.155,Z 272.592,A -85,B 0,C 180,E1 -21631.751,E2 -21631.751} C_VEL
LIN {X 0,Y 223.639,Z 278.116,A -85,B 0,C 180,E1 -21633.076,E2 -21633.076} C_VEL
LIN {X 0,Y 227.553,Z 284.895,A -85,B 0,C 180,E1 -21634.917,E2 -21634.917} C_VEL
LIN {X 0,Y 233.933,Z 296.878,A -85,B 0,C 180,E1 -21637.674,E2 -21637.674} C_VEL
LIN {X 0,Y 239.262,Z 308.198,A -85,B 0,C 180,E1 -21639.808,E2 -21639.808} C_VEL
LIN {X 0,Y 243.923,Z 319.315,A -85,B 0,C 180,E1 -21641.58,E2 -21641.58} C_VEL
LIN {X 0,Y 238.501,Z 401.677,A -85,B 0,C 180,E1 -21643.786,E2 -21643.786} C_VEL
LIN {X 0,Y 236.406,Z 417.81,A -85,B 0,C 180,E1 -21644.482,E2 -21644.482} C_VEL
LIN {X 0,Y 233.488,Z 433.053,A -85,B 0,C 180,E1 -21645.437,E2 -21645.437} C_VEL
LIN {X 0,Y 230.107,Z 446.785,A -85,B 0,C 180,E1 -21646.592,E2 -21646.592} C_VEL
LIN {X 0,Y 226.25,Z 460.166,A -85,B 0,C 180,E1 -21648.085,E2 -21648.085} C_VEL
LIN {X 0,Y 221.617,Z 473.955,A -85,B 0,C 180,E1 -21650.047,E2 -21650.047} C_VEL
LIN {X 0,Y 216.711,Z 486.369,A -85,B 0,C 180,E1 -21652.258,E2 -21652.258} C_VEL
LIN {X 0,Y 211.534,Z 498.549,A -85,B 0,C 180,E1 -21655.033,E2 -21655.033} C_VEL
LIN {X 0,Y 206.526,Z 509.31,A -85,B 0,C 180,E1 -21658.134,E2 -21658.134} C_VEL
LIN {X 0,Y 202.269,Z 518.429,A -85,B 0,C 180,E1 -21661.462,E2 -21661.462} C_VEL
LIN {X 0,Y 198.518,Z 525.931,A -85,B 0,C 180,E1 -21664.861,E2 -21664.861} C_VEL
LIN {X 0,Y 195.15,Z 532.936,A -85,B 0,C 180,E1 -21668.892,E2 -21668.892} C_VEL
LIN {X 0,Y 192.7,Z 538.451,A -85,B 0,C 180,E1 -21673.037,E2 -21673.037} C_VEL
LIN {X 0,Y 191.066,Z 542.627,A -85,B 0,C 180,E1 -21677.25,E2 -21677.25} C_VEL
LIN {X 0,Y 190.285,Z 545.563,A -85,B 0,C 180,E1 -21681.504,E2 -21681.504} C_VEL
LIN {X 0,Y 190.081,Z 547.319,A -85,B 0,C 180,E1 -21685.759,E2 -21685.759} C_VEL
LIN {X 0,Y 190.263,Z 547.924,A -85,B 0,C 180,E1 -21690,E2 -21690} C_VEL
LIN {X 0,Y 190.081,Z 547.303,A -85,B 0,C 180,E1 -21694.241,E2 -21694.241} C_VEL
LIN {X 0,Y 190.285,Z 545.527,A -85,B 0,C 180,E1 -21698.496,E2 -21698.496} C_VEL
LIN {X 0,Y 191.062,Z 542.576,A -85,B 0,C 180,E1 -21702.75,E2 -21702.75} C_VEL
LIN {X 0,Y 192.658,Z 538.385,A -85,B 0,C 180,E1 -21706.967,E2 -21706.967} C_VEL
LIN {X 0,Y 195.091,Z 532.845,A -85,B 0,C 180,E1 -21711.115,E2 -21711.115} C_VEL
LIN {X 0,Y 198.505,Z 525.81,A -85,B 0,C 180,E1 -21715.141,E2 -21715.141} C_VEL
LIN {X 0,Y 202.26,Z 518.295,A -85,B 0,C 180,E1 -21718.54,E2 -21718.54} C_VEL
LIN {X 0,Y 206.371,Z 509.442,A -85,B 0,C 180,E1 -21721.772,E2 -21721.772} C_VEL
LIN {X 0,Y 210.73,Z 499.995,A -85,B 0,C 180,E1 -21724.538,E2 -21724.538} C_VEL
LIN {X 0,Y 215.427,Z 489.115,A -85,B 0,C 180,E1 -21727.123,E2 -21727.123} C_VEL
LIN {X 0,Y 220.218,Z 477.247,A -85,B 0,C 180,E1 -21729.366,E2 -21729.366} C_VEL
LIN {X 0,Y 224.735,Z 464.41,A -85,B 0,C 180,E1 -21731.317,E2 -21731.317} C_VEL
LIN {X 0,Y 228.622,Z 451.691,A -85,B 0,C 180,E1 -21732.853,E2 -21732.853} C_VEL
LIN {X 0,Y 232.354,Z 437.038,A -85,B 0,C 180,E1 -21734.231,E2 -21734.231} C_VEL
LIN {X 0,Y 235.443,Z 422.435,A -85,B 0,C 180,E1 -21735.223,E2 -21735.223} C_VEL
LIN {X 0,Y 237.722,Z 407.486,A -85,B 0,C 180,E1 -21735.952,E2 -21735.952} C_VEL
LIN {X 0,Y 239.198,Z 390.648,A -85,B 0,C 180,E1 -21736.497,E2 -21736.497} C_VEL
LIN {X 0,Y 243.775,Z 319.188,A -85,B 0,C 180,E1 -21738.389,E2 -21738.389} C_VEL
LIN {X 0,Y 238.196,Z 305.964,A -85,B 0,C 180,E1 -21740.518,E2 -21740.518} C_VEL
LIN {X 0,Y 233.088,Z 295.419,A -85,B 0,C 180,E1 -21742.574,E2 -21742.574} C_VEL
LIN {X 0,Y 226.821,Z 283.584,A -85,B 0,C 180,E1 -21745.313,E2 -21745.313} C_VEL
LIN {X 0,Y 221.462,Z 274.466,A -85,B 0,C 180,E1 -21747.89,E2 -21747.89} C_VEL
LIN {X 0,Y 218.044,Z 269.147,A -85,B 0,C 180,E1 -21749.674,E2 -21749.674} C_VEL
LIN {X 0,Y 214.873,Z 264.951,A -85,B 0,C 180,E1 -21751.422,E2 -21751.422} C_VEL
LIN {X 0,Y 211.877,Z 261.029,A -85,B 0,C 180,E1 -21753.218,E2 -21753.218} C_VEL
LIN {X 0,Y 208.375,Z 256.904,A -85,B 0,C 180,E1 -21755.504,E2 -21755.504} C_VEL
LIN {X 0,Y 207.408,Z 255.363,A -85,B 0,C 180,E1 -21756.219,E2 -21756.219} C_VEL
LIN {X 0,Y 204.699,Z 252.891,A -85,B 0,C 180,E1 -21758.209,E2 -21758.209} C_VEL
LIN {X 0,Y 202.973,Z 249.897,A -85,B 0,C 180,E1 -21759.742,E2 -21759.742} C_VEL
LIN {X 0,Y 200.244,Z 247.959,A -85,B 0,C 180,E1 -21762.166,E2 -21762.166} C_VEL
LIN {X 0,Y 198.555,Z 245.155,A -85,B 0,C 180,E1 -21764.079,E2 -21764.079} C_VEL
LIN {X 0,Y 198.196,Z 244.127,A -85,B 0,C 180,E1 -21764.577,E2 -21764.577} C_VEL
LIN {X 0,Y 195.242,Z 242.574,A -85,B 0,C 180,E1 -21768.318,E2 -21768.318} C_VEL
LIN {X 0,Y 193.48,Z 239.818,A -85,B 0,C 180,E1 -21771.777,E2 -21771.777} C_VEL
LIN {X 0,Y 192.98,Z 238.072,A -85,B 0,C 180,E1 -21773.465,E2 -21773.465} C_VEL
LIN {X 0,Y 193.258,Z 238.038,A -85,B 0,C 180,E1 -21777.916,E2 -21777.916} C_VEL
LIN {X 0,Y 193.439,Z 238.001,A -85,B 0,C 180,E1 -21780,E2 -21780} C_VEL
LIN {X 0,Y 192.969,Z 238.06,A -85,B 0,C 180,E1 -21784.177,E2 -21784.177} C_VEL
LIN {X 0,Y 193.032,Z 238.216,A -85,B 0,C 180,E1 -21787.256,E2 -21787.256} C_VEL
LIN {X 0,Y 194.029,Z 240.994,A -85,B 0,C 180,E1 -21789.952,E2 -21789.952} C_VEL
LIN {X 0,Y 196.172,Z 243.303,A -85,B 0,C 180,E1 -21793.466,E2 -21793.466} C_VEL
LIN {X 0,Y 198.301,Z 244.39,A -85,B 0,C 180,E1 -21796.009,E2 -21796.009} C_VEL
LIN {X 0,Y 199.754,Z 247.398,A -85,B 0,C 180,E1 -21797.777,E2 -21797.777} C_VEL
LIN {X 0,Y 202.203,Z 249.557,A -85,B 0,C 180,E1 -21800.074,E2 -21800.074} C_VEL
LIN {X 0,Y 203.108,Z 250.131,A -85,B 0,C 180,E1 -21800.826,E2 -21800.826} C_VEL
LIN {X 0,Y 205.073,Z 253.376,A -85,B 0,C 180,E1 -21802.535,E2 -21802.535} C_VEL
LIN {X 0,Y 207.763,Z 255.828,A -85,B 0,C 180,E1 -21804.481,E2 -21804.481} C_VEL
LIN {X 0,Y 210.176,Z 259.263,A -85,B 0,C 180,E1 -21806.166,E2 -21806.166} C_VEL
LIN {X 0,Y 211.933,Z 261.113,A -85,B 0,C 180,E1 -21807.261,E2 -21807.261} C_VEL
LIN {X 0,Y 214.62,Z 264.723,A -85,B 0,C 180,E1 -21808.882,E2 -21808.882} C_VEL
LIN {X 0,Y 215.84,Z 266.257,A -85,B 0,C 180,E1 -21809.571,E2 -21809.571} C_VEL
LIN {X 0,Y 220.011,Z 271.892,A -85,B 0,C 180,E1 -21811.794,E2 -21811.794} C_VEL
LIN {X 0,Y 222.901,Z 275.931,A -85,B 0,C 180,E1 -21813.218,E2 -21813.218} C_VEL
LIN {X 0,Y 228.723,Z 284.486,A -85,B 0,C 180,E1 -21815.855,E2 -21815.855} C_VEL
LIN {X 0,Y 235.815,Z 295.959,A -85,B 0,C 180,E1 -21818.746,E2 -21818.746} C_VEL
LIN {X 0,Y 241.907,Z 306.998,A -85,B 0,C 180,E1 -21821.018,E2 -21821.018} C_VEL
LIN {X 0,Y 244.112,Z 312.029,A -85,B 0,C 180,E1 -21821.833,E2 -21821.833} C_VEL
LIN {X 0,Y 238.956,Z 391.512,A -85,B 0,C 180,E1 -21823.975,E2 -21823.975} C_VEL
LIN {X 0,Y 237.074,Z 407.121,A -85,B 0,C 180,E1 -21824.646,E2 -21824.646} C_VEL
LIN {X 0,Y 234.321,Z 422.708,A -85,B 0,C 180,E1 -21825.638,E2 -21825.638} C_VEL
LIN {X 0,Y 230.94,Z 437.539,A -85,B 0,C 180,E1 -21826.946,E2 -21826.946} C_VEL
LIN {X 0,Y 227.093,Z 451.6,A -85,B 0,C 180,E1 -21828.586,E2 -21828.586} C_VEL
LIN {X 0,Y 222.532,Z 465.045,A -85,B 0,C 180,E1 -21830.538,E2 -21830.538} C_VEL
LIN {X 0,Y 217.886,Z 477.244,A -85,B 0,C 180,E1 -21832.787,E2 -21832.787} C_VEL
LIN {X 0,Y 213.135,Z 488.359,A -85,B 0,C 180,E1 -21835.334,E2 -21835.334} C_VEL
LIN {X 0,Y 208.31,Z 499.141,A -85,B 0,C 180,E1 -21838.471,E2 -21838.471} C_VEL
LIN {X 0,Y 203.859,Z 508.097,A -85,B 0,C 180,E1 -21841.705,E2 -21841.705} C_VEL
